(* CoDeSys 2.3.9.50 project: 152_1sha1.pro *)
(* Libraries: STANDARD.LIB 4.10.05 11:14:46, TcBase.lib 14.5.09 12:14:08, TcSystem.lib 7.6.16 11:01:22, TcUtilities.lib 16.7.20 16:08:25, SysLibVisu.lib 7.7.04 18:17:22, SysLibTargetVisu.lib 16.6.08 16:24:26, Util.lib 18.5.10 15:14:28 *)

(* Task configuration *)
TASK Standard (PRIORITY := 0, INTERVAL := T#10ms);
	MAIN
END_TASK
TASK VISU_TASK (PRIORITY := 3, INTERVAL := T#200ms);
	MAINTARGETVISU_PAINT_CODE
END_TASK
TASK VISU_INPUT_TASK (PRIORITY := 2, INTERVAL := T#50ms);
	MAINTARGETVISU_INPUT_CODE
END_TASK

(* Global variable list: Global_Variables *)
VAR_GLOBAL
(*---------------- ЛАМПЫ -------------------*)

	K152_1SHA1_HL1 					AT %Q* 	: BOOL;			(* Сеть *)
	K152_1SHA1_HL2 					AT %Q* 	: BOOL;			(* Общая авария / авария сети *)

(*----------------СОСТОЯНИЕ АВТОМАТОВ -----------------*)

	K152_1SHA1_QF1 							AT %I* 		: BOOL;		(* Положение автоматического выключателя QF1 *)
	K152_1SHA1_SF3 							AT %I* 		: BOOL;		(* Положение автоматического выключателя SF3 *)

(*----------------РАБОТА БП----------------*)

	masTABLE_POWER 							: ARRAY [1..25] OF TABLE_POWER;

	WORK_BP 									AT %I*		: BOOL;		(* Работа БП *)
	WORK_IBP 								AT %I*		: BOOL;		(* Работа ИБП *)
	WORK_OF_BATTERY 						AT %I*		: BOOL;		(* Работа от батареи *)
	REPLACE_BATTERY 						AT %I*		: BOOL;		(* Замените батарею *)

	K152_1SHA1_WORK_BP 					AT %Q*		: BOOL;		(* Работа БП *)
	K152_1SHA1_WORK_IBP 					AT %Q*		: BOOL;		(* Работа ИБП *)
	K152_1SHA1_WORK_OF_BATTERY 		AT %Q*		: BOOL;		(* Работа от батареи *)
	K152_1SHA1_REPLACE_BATTERY 			AT %Q*		: BOOL;		(* Замените батарею *)

(*---------------- ЩАО1 ----------------*)

	K152_1SHA1_SCHAO1_POWER			AT %I*		: BOOL;		(* Наличие напряжения на вводе *)
	K152_1SHA1_SCHAO1_QF1				AT %I*		: BOOL;		(* Включен автоматический выключатель QF1 *)
	K152_1SHA1_SCHAO1_QF2				AT %I*		: BOOL;		(* Включен автоматический выключатель QF2 *)
	K152_1SHA1_SCHAO1_QF3				AT %I*		: BOOL;		(* Включен автоматический выключатель QF3 *)
	K152_1SHA1_SCHAO1_QF4				AT %I*		: BOOL;		(* Включен автоматический выключатель QF4 *)
	K152_1SHA1_SCHAO1_QF5				AT %I*		: BOOL;		(* Включен автоматический выключатель QF5 *)
	K152_1SHA1_SCHAO1_QF6				AT %I*		: BOOL;		(* Включен автоматический выключатель QF6 *)
	K152_1SHA1_SCHAO1_QF7				AT %I*		: BOOL;		(* Включен автоматический выключатель QF7 *)

	K152_1SHA1_SCHAO1_KM_GR5			AT %I*		: BOOL;		(* Положение магнитного пускателя гр.5 *)

	K152_1SHA1_SCHAO1_SA_AVT_GR5		AT %I*		: BOOL;		(* Положение переключателя в режиме Авт. гр.5 *)
	K152_1SHA1_SCHAO1_SA_RUCH_GR5		AT %I*		: BOOL;		(* ?????	СМ	СХЕМУ		???????? Положение переключателя в режиме Руч. гр.5 *)

	bK152_1SHA1_SCHAO1_LIGHT_GR5_ON				: BOOL;		(* Кнопка включения группы освещения. гр.5 *)
	bK152_1SHA1_SCHAO1_LIGHT_GR5_OFF				: BOOL;		(* Кнопка выключения группы освещения. гр.5 *)
	K152_1SHA1_SCHAO1_LIGHT_GR5			AT %Q*		: BOOL;		(* Сигнал на включение группы освещения. гр.5 *)

	masTABLE_SCHAO1									: ARRAY [1..11] OF TABLE_SCHAO1;

	st_SCHAO1_POWER									: STRING;		(* Наличие напряжения на вводе *)
	st_SCHAO1_QF1										: STRING;		(* Включен автоматический выключатель QF1 *)
	st_SCHAO1_QF2										: STRING;		(* Включен автоматический выключатель QF2 *)
	st_SCHAO1_QF3										: STRING;		(* Включен автоматический выключатель QF3 *)
	st_SCHAO1_QF4										: STRING;		(* Включен автоматический выключатель QF4 *)
	st_SCHAO1_QF5										: STRING;		(* Включен автоматический выключатель QF5 *)
	st_SCHAO1_QF6										: STRING;		(* Включен автоматический выключатель QF6 *)
	st_SCHAO1_QF7										: STRING;		(* Включен автоматический выключатель QF7 *)

	st_SCHAO1_KM_GR5									: STRING;		(* Положение магнитного пускателя гр.5 *)

	st_SCHAO1_SA_AVT_GR5								: STRING;		(* Положение переключателя в режиме Авт. гр.5 *)
	st_SCHAO1_SA_RUCH_GR5							: STRING;		(* ?????	СМ	СХЕМУ		???????? Положение переключателя в режиме Руч. гр.5 *)

	st_SCHAO1_LIGHT_GR5								: STRING;		(* Сигнал на включение группы освещения. гр.5 *)

(*---------------- ЩАО2 ----------------*)

	K152_1SHA1_SCHAO2_POWER			AT %I*		: BOOL;		(* Наличие напряжения на вводе *)
	K152_1SHA1_SCHAO2_QF1				AT %I*		: BOOL;		(* Включен автоматический выключатель QF1 *)
	K152_1SHA1_SCHAO2_QF2				AT %I*		: BOOL;		(* Включен автоматический выключатель QF2 *)
	K152_1SHA1_SCHAO2_QF3				AT %I*		: BOOL;		(* Включен автоматический выключатель QF3 *)
	K152_1SHA1_SCHAO2_QF4				AT %I*		: BOOL;		(* Включен автоматический выключатель QF4 *)
	K152_1SHA1_SCHAO2_QF5				AT %I*		: BOOL;		(* Включен автоматический выключатель QF5 *)
	K152_1SHA1_SCHAO2_QF6				AT %I*		: BOOL;		(* Включен автоматический выключатель QF6 *)
	K152_1SHA1_SCHAO2_QF7				AT %I*		: BOOL;		(* Включен автоматический выключатель QF7 *)
	K152_1SHA1_SCHAO2_QF8				AT %I*		: BOOL;		(* Включен автоматический выключатель QF8 *)
	K152_1SHA1_SCHAO2_QF9				AT %I*		: BOOL;		(* Включен автоматический выключатель QF9 *)

	K152_1SHA1_SCHAO2_KM_GR5			AT %I*		: BOOL;		(* Положение магнитного пускателя гр.5 *)

	K152_1SHA1_SCHAO2_SA_AVT_GR5		AT %I*		: BOOL;		(* Положение переключателя в режиме Авт. гр.5 *)
	K152_1SHA1_SCHAO2_SA_RUCH_GR5		AT %I*		: BOOL;		(* ?????	СМ	СХЕМУ		???????? Положение переключателя в режиме Руч. гр.5 *)

	K152_1SHA1_SCHAO2_LIGHT_GR5			AT %Q*		: BOOL;		(* Сигнал на включение группы освещения. гр.5 *)

	masTABLE_SCHAO2									: ARRAY [1..13] OF TABLE_SCHAO2;

	st_SCHAO2_POWER									: STRING;		(* Наличие напряжения на вводе *)
	st_SCHAO2_QF1										: STRING;		(* Включен автоматический выключатель QF1 *)
	st_SCHAO2_QF2										: STRING;		(* Включен автоматический выключатель QF2 *)
	st_SCHAO2_QF3										: STRING;		(* Включен автоматический выключатель QF3 *)
	st_SCHAO2_QF4										: STRING;		(* Включен автоматический выключатель QF4 *)
	st_SCHAO2_QF5										: STRING;		(* Включен автоматический выключатель QF5 *)
	st_SCHAO2_QF6										: STRING;		(* Включен автоматический выключатель QF6 *)
	st_SCHAO2_QF7										: STRING;		(* Включен автоматический выключатель QF7 *)
	st_SCHAO2_QF8										: STRING;		(* Включен автоматический выключатель QF8 *)
	st_SCHAO2_QF9										: STRING;		(* Включен автоматический выключатель QF9 *)

	st_SCHAO2_KM_GR5									: STRING;		(* Положение магнитного пускателя гр.5 *)

	st_SCHAO2_SA_AVT_GR5								: STRING;		(* Положение переключателя в режиме Авт. гр.5 *)
	st_SCHAO2_SA_RUCH_GR5							: STRING;		(* ?????	СМ	СХЕМУ		???????? Положение переключателя в режиме Руч. гр.5 *)

	st_SCHAO2_LIGHT_GR5								: STRING;		(* Сигнал на включение группы освещения. гр.5 *)

	bK152_1SHA1_SCHAO2_LIGHT_GR5_ON				: BOOL;		(* Кнопка включения группы освещения. гр.5 *)
	bK152_1SHA1_SCHAO2_LIGHT_GR5_OFF				: BOOL;		(* Кнопка выключения группы освещения. гр.5 *)

(*---------------- ЩО1 ----------------*)

	K152_1SHA1_SCHO1_QF1					AT %I*		: BOOL;		(* Включен автоматический выключатель QF1 *)
	K152_1SHA1_SCHO1_QF2					AT %I*		: BOOL;		(* Включен автоматический выключатель QF2 *)

	K152_1SHA1_SCHO1_KM_GR1				AT %I*		: BOOL;		(* Положение магнитного пускателя гр.1 *)
	K152_1SHA1_SCHO1_KM_GR2				AT %I*		: BOOL;		(* Положение магнитного пускателя гр.2 *)

	K152_1SHA1_SCHO1_SA_AVT_GR1		AT %I*		: BOOL;		(* Положение переключателя в режиме Авт. гр.1 *)
	K152_1SHA1_SCHO1_SA_AVT_GR2		AT %I*		: BOOL;		(* Положение переключателя в режиме Авт. гр.2 *)

	K152_1SHA1_SCHO1_SA_RUCH_GR1		AT %I*		: BOOL;		(* Положение переключателя в режиме Руч. гр.1 *)
	K152_1SHA1_SCHO1_SA_RUCH_GR2		AT %I*		: BOOL;		(* Положение переключателя в режиме Руч. гр.2 *)

	K152_1SHA1_SCHO1_LIGHT_GR1			AT %Q*		: BOOL;		(* Сигнал на включение группы освещения. гр.1 *)
	K152_1SHA1_SCHO1_LIGHT_GR2			AT %Q*		: BOOL;		(* Сигнал на включение группы освещения. гр.2 *)

	masTABLE_SCHO1										: ARRAY [1..8] OF TABLE_SCHO1;

	st_SCHO1_QF1											: STRING;		(* Включен автоматический выключатель QF1 *)
	st_SCHO1_QF2											: STRING;		(* Включен автоматический выключатель QF2 *)

	st_SCHO1_KM_GR1									: STRING;		(* Положение магнитного пускателя гр.1 *)
	st_SCHO1_KM_GR2									: STRING;		(* Положение магнитного пускателя гр.2 *)

	st_SCHO1_SA_AVT_GR1								: STRING;		(* Положение переключателя в режиме Авт. гр.1 *)
	st_SCHO1_SA_AVT_GR2								: STRING;		(* Положение переключателя в режиме Авт. гр.2 *)

	st_SCHO1_SA_RUCH_GR1								: STRING;		(* Положение переключателя в режиме Руч. гр.1 *)
	st_SCHO1_SA_RUCH_GR2								: STRING;		(* Положение переключателя в режиме Руч. гр.2 *)

	st_SCHO1_LIGHT_GR1									: STRING;		(* Сигнал на включение группы освещения. гр.1 *)
	st_SCHO1_LIGHT_GR2									: STRING;		(* Сигнал на включение группы освещения. гр.2 *)

	bK152_1SHA1_SCHO1_LIGHT_GR1_ON					: BOOL;		(* Кнопка включения группы освещения. гр.1 *)
	bK152_1SHA1_SCHO1_LIGHT_GR2_ON					: BOOL;		(* Кнопка включения группы освещения. гр.2 *)
	bK152_1SHA1_SCHO1_LIGHT_GR1_OFF				: BOOL;		(* Кнопка выключения группы освещения. гр.1 *)
	bK152_1SHA1_SCHO1_LIGHT_GR2_OFF				: BOOL;		(* Кнопка выключения группы освещения. гр.2 *)

(*---------------- ЩО2 ----------------*)

	K152_1SHA1_SCHO2_QF1					AT %I*		: BOOL;		(* Включен автоматический выключатель QF1 *)
	K152_1SHA1_SCHO2_QF2					AT %I*		: BOOL;		(* Включен автоматический выключатель QF2 *)
	K152_1SHA1_SCHO2_QF3					AT %I*		: BOOL;		(* Включен автоматический выключатель QF3 *)
	K152_1SHA1_SCHO2_QF4					AT %I*		: BOOL;		(* Включен автоматический выключатель QF4 *)
	K152_1SHA1_SCHO2_QF5					AT %I*		: BOOL;		(* Включен автоматический выключатель QF5 *)
	K152_1SHA1_SCHO2_QF9					AT %I*		: BOOL;		(* Включен автоматический выключатель QF9 *)

	K152_1SHA1_SCHO2_KM_GR1				AT %I*		: BOOL;		(* Положение магнитного пускателя гр.1 *)
	K152_1SHA1_SCHO2_KM_GR2				AT %I*		: BOOL;		(* Положение магнитного пускателя гр.2 *)
	K152_1SHA1_SCHO2_KM_GR3				AT %I*		: BOOL;		(* Положение магнитного пускателя гр.3 *)
	K152_1SHA1_SCHO2_KM_GR4				AT %I*		: BOOL;		(* Положение магнитного пускателя гр.4 *)
	K152_1SHA1_SCHO2_KM_GR5				AT %I*		: BOOL;		(* Положение магнитного пускателя гр.5 *)
	K152_1SHA1_SCHO2_KM_GR9				AT %I*		: BOOL;		(* Положение магнитного пускателя гр.9 *)

	K152_1SHA1_SCHO2_SA_AVT_GR1		AT %I*		: BOOL;		(* Положение переключателя в режиме Авт. гр.1 *)
	K152_1SHA1_SCHO2_SA_AVT_GR2		AT %I*		: BOOL;		(* Положение переключателя в режиме Авт. гр.2 *)
	K152_1SHA1_SCHO2_SA_AVT_GR3		AT %I*		: BOOL;		(* Положение переключателя в режиме Авт. гр.3 *)
	K152_1SHA1_SCHO2_SA_AVT_GR4		AT %I*		: BOOL;		(* Положение переключателя в режиме Авт. гр.4 *)
	K152_1SHA1_SCHO2_SA_AVT_GR5		AT %I*		: BOOL;		(* Положение переключателя в режиме Авт. гр.5 *)
	K152_1SHA1_SCHO2_SA_AVT_GR9		AT %I*		: BOOL;		(* Положение переключателя в режиме Авт. гр.9 *)

	K152_1SHA1_SCHO2_SA_RUCH_GR1		AT %I*		: BOOL;		(* Положение переключателя в режиме Руч. гр.1 *)
	K152_1SHA1_SCHO2_SA_RUCH_GR2		AT %I*		: BOOL;		(* Положение переключателя в режиме Руч. гр.2 *)
	K152_1SHA1_SCHO2_SA_RUCH_GR3		AT %I*		: BOOL;		(* Положение переключателя в режиме Руч. гр.3 *)
	K152_1SHA1_SCHO2_SA_RUCH_GR4		AT %I*		: BOOL;		(* Положение переключателя в режиме Руч. гр.4 *)
	K152_1SHA1_SCHO2_SA_RUCH_GR5		AT %I*		: BOOL;		(* Положение переключателя в режиме Руч. гр.5 *)
	K152_1SHA1_SCHO2_SA_RUCH_GR9		AT %I*		: BOOL;		(* Положение переключателя в режиме Руч. гр.9 *)

	K152_1SHA1_SCHO2_LIGHT_GR1			AT %Q*		: BOOL;		(* Сигнал на включение группы освещения. гр.1 *)
	K152_1SHA1_SCHO2_LIGHT_GR2			AT %Q*		: BOOL;		(* Сигнал на включение группы освещения. гр.2 *)
	K152_1SHA1_SCHO2_LIGHT_GR3			AT %Q*		: BOOL;		(* Сигнал на включение группы освещения. гр.3 *)
	K152_1SHA1_SCHO2_LIGHT_GR4			AT %Q*		: BOOL;		(* Сигнал на включение группы освещения. гр.4 *)
	K152_1SHA1_SCHO2_LIGHT_GR5			AT %Q*		: BOOL;		(* Сигнал на включение группы освещения. гр.5 *)
	K152_1SHA1_SCHO2_LIGHT_GR9			AT %Q*		: BOOL;		(* Сигнал на включение группы освещения. гр.9 *)

	masTABLE_SCHO2_1									: ARRAY [1..4] OF TABLE;
	masTABLE_SCHO2_2									: ARRAY [1..4] OF TABLE_SCHO2;
	masTABLE_SCHO2_3									: ARRAY [1..4] OF TABLE_SCHO2;
	masTABLE_SCHO2_4									: ARRAY [1..4] OF TABLE_SCHO2;
	masTABLE_SCHO2_5									: ARRAY [1..4] OF TABLE_SCHO2;
	masTABLE_SCHO2_9									: ARRAY [1..4] OF TABLE_SCHO2;

	st_SCHO2_QF1											: STRING;		(* Включен автоматический выключатель QF1 *)
	st_SCHO2_QF2											: STRING;		(* Включен автоматический выключатель QF2 *)
	st_SCHO2_QF3											: STRING;		(* Включен автоматический выключатель QF3 *)
	st_SCHO2_QF4											: STRING;		(* Включен автоматический выключатель QF4 *)
	st_SCHO2_QF5											: STRING;		(* Включен автоматический выключатель QF5 *)
	st_SCHO2_QF9											: STRING;		(* Включен автоматический выключатель QF9 *)

	st_SCHO2_KM_GR1									: STRING;		(* Положение магнитного пускателя гр.1 *)
	st_SCHO2_KM_GR2									: STRING;		(* Положение магнитного пускателя гр.2 *)
	st_SCHO2_KM_GR3									: STRING;		(* Положение магнитного пускателя гр.3 *)
	st_SCHO2_KM_GR4									: STRING;		(* Положение магнитного пускателя гр.4 *)
	st_SCHO2_KM_GR5									: STRING;		(* Положение магнитного пускателя гр.5 *)
	st_SCHO2_KM_GR9									: STRING;		(* Положение магнитного пускателя гр.9 *)

	st_SCHO2_SA_AVT_GR1								: STRING;		(* Положение переключателя в режиме Авт. гр.1 *)
	st_SCHO2_SA_AVT_GR2								: STRING;		(* Положение переключателя в режиме Авт. гр.2 *)
	st_SCHO2_SA_AVT_GR3								: STRING;		(* Положение переключателя в режиме Авт. гр.3 *)
	st_SCHO2_SA_AVT_GR4								: STRING;		(* Положение переключателя в режиме Авт. гр.4 *)
	st_SCHO2_SA_AVT_GR5								: STRING;		(* Положение переключателя в режиме Авт. гр.5 *)
	st_SCHO2_SA_AVT_GR9								: STRING;		(* Положение переключателя в режиме Авт. гр.9 *)

	st_SCHO2_SA_RUCH_GR1								: STRING;		(* Положение переключателя в режиме Руч. гр.1 *)
	st_SCHO2_SA_RUCH_GR2								: STRING;		(* Положение переключателя в режиме Руч. гр.2 *)
	st_SCHO2_SA_RUCH_GR3								: STRING;		(* Положение переключателя в режиме Руч. гр.3 *)
	st_SCHO2_SA_RUCH_GR4								: STRING;		(* Положение переключателя в режиме Руч. гр.4 *)
	st_SCHO2_SA_RUCH_GR5								: STRING;		(* Положение переключателя в режиме Руч. гр.5 *)
	st_SCHO2_SA_RUCH_GR9								: STRING;		(* Положение переключателя в режиме Руч. гр.9 *)

	st_SCHO2_LIGHT_GR1									: STRING;		(* Сигнал на включение группы освещения. гр.1 *)
	st_SCHO2_LIGHT_GR2									: STRING;		(* Сигнал на включение группы освещения. гр.2 *)
	st_SCHO2_LIGHT_GR3									: STRING;		(* Сигнал на включение группы освещения. гр.3 *)
	st_SCHO2_LIGHT_GR4									: STRING;		(* Сигнал на включение группы освещения. гр.4 *)
	st_SCHO2_LIGHT_GR5									: STRING;		(* Сигнал на включение группы освещения. гр.5 *)
	st_SCHO2_LIGHT_GR9									: STRING;		(* Сигнал на включение группы освещения. гр.9 *)

	bK152_1SHA1_SCHO2_LIGHT_GR1_ON					: BOOL;		(* Кнопка включения группы освещения. гр.1 *)
	bK152_1SHA1_SCHO2_LIGHT_GR2_ON					: BOOL;		(* Кнопка включения группы освещения. гр.2 *)
	bK152_1SHA1_SCHO2_LIGHT_GR3_ON					: BOOL;		(* Кнопка включения группы освещения. гр.3 *)
	bK152_1SHA1_SCHO2_LIGHT_GR4_ON					: BOOL;		(* Кнопка включения группы освещения. гр.4 *)
	bK152_1SHA1_SCHO2_LIGHT_GR5_ON					: BOOL;		(* Кнопка включения группы освещения. гр.5 *)
	bK152_1SHA1_SCHO2_LIGHT_GR9_ON					: BOOL;		(* Кнопка включения группы освещения. гр.9 *)

	bK152_1SHA1_SCHO2_LIGHT_GR1_OFF				: BOOL;		(* Кнопка выключения группы освещения. гр.1 *)
	bK152_1SHA1_SCHO2_LIGHT_GR2_OFF				: BOOL;		(* Кнопка выключения группы освещения. гр.2 *)
	bK152_1SHA1_SCHO2_LIGHT_GR3_OFF				: BOOL;		(* Кнопка выключения группы освещения. гр.3 *)
	bK152_1SHA1_SCHO2_LIGHT_GR4_OFF				: BOOL;		(* Кнопка выключения группы освещения. гр.4 *)
	bK152_1SHA1_SCHO2_LIGHT_GR5_OFF				: BOOL;		(* Кнопка выключения группы освещения. гр.5 *)
	bK152_1SHA1_SCHO2_LIGHT_GR9_OFF				: BOOL;		(* Кнопка выключения группы освещения. гр.9 *)

(* 	Режимы работы *)
	K152_1SHA1_SCHO2_GR1_bMode		 				: BOOL;		(* Выбор режима управления Группой 1 *)
	K152_1SHA1_SCHO2_GR1_Mode		 				: STRING;		(* Режим управления Группой 1 *)

	Invisible_GR1_bMode									: BOOL;		(* Невидимость кнопок выбора режима Гр.1 *)
	Invisible_GR1_bMode_MU								: BOOL;		(* Невидимость кнопок управления руч. режима Гр.1 *)


	K152_1SHA1_SCHO2_GR1_bMode_AVT 				: BOOL;		(* Режим автоматического управления Группой 1 *)
	K152_1SHA1_SCHO2_GR2_bMode_AVT 				: BOOL;		(* Режим автоматического управления Группой 2 *)
	K152_1SHA1_SCHO2_GR3_bMode_AVT 				: BOOL;		(* Режим автоматического управления Группой 3 *)
	K152_1SHA1_SCHO2_GR4_bMode_AVT 				: BOOL;		(* Режим автоматического управления Группой 4 *)
	K152_1SHA1_SCHO2_GR5_bMode_AVT 				: BOOL;		(* Режим автоматического управления Группой 5 *)
	K152_1SHA1_SCHO2_GR9_bMode_AVT 				: BOOL;		(* Режим автоматического управления Группой 9 *)

	K152_1SHA1_SCHO2_GR1_bMode_MU	 				: BOOL;		(* Режим ручного управления Группой 1 *)
	K152_1SHA1_SCHO2_GR2_bMode_MU	 				: BOOL;		(* Режим ручного управления Группой 2 *)
	K152_1SHA1_SCHO2_GR3_bMode_MU	 				: BOOL;		(* Режим ручного управления Группой 3 *)
	K152_1SHA1_SCHO2_GR4_bMode_MU	 				: BOOL;		(* Режим ручного управления Группой 4 *)
	K152_1SHA1_SCHO2_GR5_bMode_MU	 				: BOOL;		(* Режим ручного управления Группой 5 *)
	K152_1SHA1_SCHO2_GR9_bMode_MU	 				: BOOL;		(* Режим ручного управления Группой 9 *)

(* 	Недельный график *)
	masTABLE_WEEKLY_SCHO2_GR1						: ARRAY [1..2] OF TABLE_WEEKLY_SCHEDULE;

(*---------------- Датчики протечки ----------------*)

	K152_1SHA1_LS_ITP_1						AT %I*		: BOOL;		(* Датчик протечки LS-ИТП-1 *)
	K152_1SHA1_LS_ITP_2						AT %I*		: BOOL;		(* Датчик протечки LS-ИТП-2 *)
	K152_1SHA1_LS_NS_1						AT %I*		: BOOL;		(* Датчик протечки LS-НС-1 *)
	K152_1SHA1_LS_NS_2						AT %I*		: BOOL;		(* Датчик протечки LS-НС-2 *)

(*---------------- Коробка соединительная КС1 ----------------*)

	K152_1SHA1_KC1_BK1_TRESH1			AT %I*		: BOOL;		(* Блок контроля 1, Срабатывание порога 1 *)
	K152_1SHA1_KC1_BK2_TRESH1			AT %I*		: BOOL;		(* Блок контроля 2, Срабатывание порога 1 *)
	K152_1SHA1_KC1_BK3_TRESH1			AT %I*		: BOOL;		(* Блок контроля 3, Срабатывание порога 1 *)
	K152_1SHA1_KC1_BK4_TRESH1			AT %I*		: BOOL;		(* Блок контроля 4, Срабатывание порога 1 *)

	K152_1SHA1_KC1_BK1_TRESH2			AT %I*		: BOOL;		(* Блок контроля 1, Срабатывание порога 2 *)
	K152_1SHA1_KC1_BK2_TRESH2			AT %I*		: BOOL;		(* Блок контроля 2, Срабатывание порога 2 *)
	K152_1SHA1_KC1_BK3_TRESH2			AT %I*		: BOOL;		(* Блок контроля 3, Срабатывание порога 2 *)
	K152_1SHA1_KC1_BK4_TRESH2			AT %I*		: BOOL;		(* Блок контроля 4, Срабатывание порога 2 *)

	K152_1SHA1_KC1_BLIND_CLOSE			AT %Q*		: BOOL;		(* Сигнал на закрытие жалюзи помещение 1.4.2 *)
	K152_1SHA1_KC1_BLIND_OPEN			AT %Q*		: BOOL;		(* Сигнал на открытие жалюзи помещение 1.4.2 *)

(*---------------- Коробка соединительная КС2 ----------------*)

	K152_1SHA1_KC2_BLIND_CLOSE			AT %Q*		: BOOL;		(* Сигнал на закрытие жалюзи помещение 1.4.1 *)
	K152_1SHA1_KC2_BLIND_OPEN			AT %Q*		: BOOL;		(* Сигнал на открытие жалюзи помещение 1.4.1 *)

(*---------------- Коробка соединительная КС3 ----------------*)

	K152_1SHA1_KC3_BLIND_CLOSE			AT %Q*		: BOOL;		(* Сигнал на закрытие жалюзи помещение 1.4.0 *)
	K152_1SHA1_KC3_BLIND_OPEN			AT %Q*		: BOOL;		(* Сигнал на открытие жалюзи помещение 1.4.0 *)

(*---------------- ШРС ----------------*)

	K152_1SHA1_WORK_ALARM_MEDOMAT	AT %I*		: BOOL;		(* Контроль работы / аварии установки Medomat *)
	K152_1SHA1_WORK_ALARM_FILTER1		AT %I*		: BOOL;		(* Контроль работы / аварии фильтра обезжелезивания 1 *)
	K152_1SHA1_WORK_ALARM_FILTER2		AT %I*		: BOOL;		(* Контроль работы / аварии фильтра обезжелезивания 2 *)
	K152_1SHA1_WORK_ALARM_RONDOMAT	AT %I*		: BOOL;		(* Контроль работы / аварии установки Rondomat *)

 	K152_1SHA1_LEVEL_TANK1				AT %I*		: BOOL;		(* Контроль уровня жидкости в резервуре 1 *)
 	K152_1SHA1_LEVEL_TANK2				AT %I*		: BOOL;		(* Контроль уровня жидкости в резервуре 2 *)
 	K152_1SHA1_LEVEL_TANK3				AT %I*		: BOOL;		(* Контроль уровня жидкости в резервуре 3 *)
 	K152_1SHA1_LEVEL_TANK4				AT %I*		: BOOL;		(* Контроль уровня жидкости в резервуре 4 *)
 	K152_1SHA1_LEVEL_TANK5				AT %I*		: BOOL;		(* Контроль уровня жидкости в резервуре 5 *)

 	K152_1SHA1_WORK_ALARM_OSMOSIS	AT %I*		: BOOL;		(* Контроль работы / аварии установки обратного осмоса *)

(*---------------- ПКУ1 ----------------*)

	K152_1SHA1_PKU1_SA					AT %I*		: BOOL;		(* Переключатель руч. / авт. помещение 1.4.2 *)
	K152_1SHA1_PKU1_SB_CLOSE			AT %I*		: BOOL;		(* Кнопка закрыть жалюзи помещение 1.4.2 *)
	K152_1SHA1_PKU1_SB_OPEN				AT %I*		: BOOL;		(* Кнопка открыть жалюзи помещение 1.4.2 *)

(*---------------- ПКУ2 ----------------*)

	K152_1SHA1_PKU2_SA					AT %I*		: BOOL;		(* Переключатель руч. / авт. помещение 1.4.1 *)
	K152_1SHA1_PKU2_SB_CLOSE			AT %I*		: BOOL;		(* Кнопка закрыть жалюзи помещение 1.4.1 *)
	K152_1SHA1_PKU2_SB_OPEN				AT %I*		: BOOL;		(* Кнопка открыть жалюзи помещение 1.4.1 *)

(*---------------- ПКУ3 ----------------*)

	K152_1SHA1_PKU3_SA					AT %I*		: BOOL;		(* Переключатель руч. / авт. помещение 1.4.0 *)
	K152_1SHA1_PKU3_SB_CLOSE			AT %I*		: BOOL;		(* Кнопка закрыть жалюзи помещение 1.4.0 *)
	K152_1SHA1_PKU3_SB_OPEN				AT %I*		: BOOL;		(* Кнопка открыть жалюзи помещение 1.4.0 *)

(*----------------ТЕМПЕРАТУРА----------------*)

	masTABLE_TEMPERATURE					: ARRAY [1..10] OF TABLE_TEMPERATURE;

	TE_TK 										AT %I*		: INT;			(* Температура воздуха в ТК, TE-TK *)
	TE_GRSCHA 								AT %I*		: INT;			(* Температура воздуха в ГРЩ TE-ГРЩ *)

	K152_1SHA1_TE_TK 						AT %Q*		: REAL;			(* Температура воздуха в ТК, TE-TK *)
	K152_1SHA1_TE_GRSCHA					AT %Q*		: REAL;			(* Температура воздуха в ГРЩ, TE-ГРЩ *)


(* --------------------- СИСТЕМНОЕ ДАТА И ВРЕМЯ -------------------------- *)
	stDate 													: STRING;		(* Текущая дата *)
	stTime 													: STRING;		(* Текущее время *)
	stTime_graphic											: STRING;		(* Часы и минуты для недельного графика *)

	Day_of_Today											: STRING;		(* Текущий день недели *)
(* --------------------- ТАБЛИЦА АВАРИЙ -------------------------- *)

	(* Дата и время *)
	stTime_Alarm											: STRING;
	stDate_Alarm											: STRING;

	(* --------------------- *)
(*
	rt_K152_1ITP_K1 								: R_TRIG ;			(* Авария входного напряжения *)
	ft_K152_1ITP_1PDS1 							: F_TRIG;			(* Перепад давления в системе отопления *)
	ft_K152_1ITP_2PDS1 							: F_TRIG;			(* Перепад давления в системе ГВС *)
	ft_K152_1ITP_2PDS2 							: F_TRIG;			(* Перепад давления в системе вентиляции *)
	ft_K152_1ITP_2PDS3 							: F_TRIG;			(* Перепад давления в системе подпитки вентиляции *)
	rt_K152_1ITP_QF1_ALARM 						: R_TRIG;
	rt_K152_1ITP_QF2_ALARM 						: R_TRIG;
	rt_K152_1ITP_QF3_ALARM	 					: R_TRIG;
	rt_K152_1ITP_QF4_ALARM 						: R_TRIG;
	rt_K152_1ITP_QF5_ALARM 						: R_TRIG;
	rt_K152_1ITP_QF6_ALARM 						: R_TRIG;
	rt_K152_1ITP_QF7_ALARM 						: R_TRIG;
	rt_K152_1ITP_QF8_ALARM 						: R_TRIG;

	rt_K152_1ITP_REPLACE_BATTERY				: R_TRIG;

	rt_K152_1ITP_UPK_ALARM 					: R_TRIG;			(* Авария установки перекачки конденсата *)
	rt_K152_1ITP_LS 								: R_TRIG;			(* Низкий уровень воды в баке ресивере *)

	rt_K152_1ITP_HL4 								: R_TRIG;			(* Авария основного насоса 2.1 *)
	rt_K152_1ITP_HL6 								: R_TRIG;			(* Авария резервного насоса 2.2 *)
	rt_K152_1ITP_HL8 								: R_TRIG;			(* Авария основного насоса 6.1 *)
	rt_K152_1ITP_HL10 								: R_TRIG;			(* Авария резервного насоса 6.2 *)
	rt_K152_1ITP_HL12 								: R_TRIG;			(* Авария основного насоса 7.1 *)
	rt_K152_1ITP_HL14 								: R_TRIG;			(* Авария резервного насоса 7.2 *)
	rt_K152_1ITP_HL16 								: R_TRIG;			(* Авария основного насоса 12.1 *)
	rt_K152_1ITP_HL18 								: R_TRIG;			(* Авария резервного насоса 12.2 *)
*)
	i 												: INT 	:= 	0;		(* Счетчик строк в таблице аварий *)
	d 												: INT 	:= 	0;		(* Счетчик записей в массив данных об авариях *)

	ALARM_TABLE 								: ARRAY [1..23] OF TABLE_ALARM;
	ALARM_DATA 									: ARRAY [1..100] OF STRING;					(* Запись инфо об аварии в одну переменную *)

	bClearAlarmData 								: BOOL;
	rt_bClearAlarmData								: R_TRIG;

END_VAR

(* Global variable list: TwinCAT_Configuration *)
(* Generated automatically by TwinCAT - (read only) *)
VAR_CONFIG
	.K152_1SHA1_HL1 AT %QX12.0 : BOOL;
	.K152_1SHA1_HL2 AT %QX12.1 : BOOL;
	.K152_1SHA1_QF1 AT %IX4.0 : BOOL;
	.K152_1SHA1_SF3 AT %IX4.1 : BOOL;
	.WORK_BP AT %IX4.2 : BOOL;
	.WORK_IBP AT %IX4.3 : BOOL;
	.WORK_OF_BATTERY AT %IX4.4 : BOOL;
	.REPLACE_BATTERY AT %IX4.5 : BOOL;
	.K152_1SHA1_WORK_BP AT %QX8.0 : BOOL;
	.K152_1SHA1_WORK_IBP AT %QX8.1 : BOOL;
	.K152_1SHA1_WORK_OF_BATTERY AT %QX8.2 : BOOL;
	.K152_1SHA1_REPLACE_BATTERY AT %QX8.3 : BOOL;
	.K152_1SHA1_SCHAO1_POWER AT %IX4.6 : BOOL;
	.K152_1SHA1_SCHAO1_QF1 AT %IX4.7 : BOOL;
	.K152_1SHA1_SCHAO1_QF2 AT %IX5.0 : BOOL;
	.K152_1SHA1_SCHAO1_QF3 AT %IX5.1 : BOOL;
	.K152_1SHA1_SCHAO1_QF4 AT %IX5.2 : BOOL;
	.K152_1SHA1_SCHAO1_QF5 AT %IX5.3 : BOOL;
	.K152_1SHA1_SCHAO1_QF6 AT %IX5.4 : BOOL;
	.K152_1SHA1_SCHAO1_QF7 AT %IX5.5 : BOOL;
	.K152_1SHA1_SCHAO1_KM_GR5 AT %IX5.6 : BOOL;
	.K152_1SHA1_SCHAO1_SA_AVT_GR5 AT %IX5.7 : BOOL;
	.K152_1SHA1_SCHAO1_SA_RUCH_GR5 AT %IX6.0 : BOOL;
	.K152_1SHA1_SCHAO1_LIGHT_GR5 AT %QX8.4 : BOOL;
	.K152_1SHA1_SCHAO2_POWER AT %IX6.1 : BOOL;
	.K152_1SHA1_SCHAO2_QF1 AT %IX6.2 : BOOL;
	.K152_1SHA1_SCHAO2_QF2 AT %IX6.3 : BOOL;
	.K152_1SHA1_SCHAO2_QF3 AT %IX6.4 : BOOL;
	.K152_1SHA1_SCHAO2_QF4 AT %IX6.5 : BOOL;
	.K152_1SHA1_SCHAO2_QF5 AT %IX6.6 : BOOL;
	.K152_1SHA1_SCHAO2_QF6 AT %IX6.7 : BOOL;
	.K152_1SHA1_SCHAO2_QF7 AT %IX7.0 : BOOL;
	.K152_1SHA1_SCHAO2_QF8 AT %IX7.1 : BOOL;
	.K152_1SHA1_SCHAO2_QF9 AT %IX7.2 : BOOL;
	.K152_1SHA1_SCHAO2_KM_GR5 AT %IX7.3 : BOOL;
	.K152_1SHA1_SCHAO2_SA_AVT_GR5 AT %IX7.4 : BOOL;
	.K152_1SHA1_SCHAO2_SA_RUCH_GR5 AT %IX7.5 : BOOL;
	.K152_1SHA1_SCHAO2_LIGHT_GR5 AT %QX8.5 : BOOL;
	.K152_1SHA1_SCHO1_QF1 AT %IX7.6 : BOOL;
	.K152_1SHA1_SCHO1_QF2 AT %IX7.7 : BOOL;
	.K152_1SHA1_SCHO1_KM_GR1 AT %IX8.0 : BOOL;
	.K152_1SHA1_SCHO1_KM_GR2 AT %IX8.1 : BOOL;
	.K152_1SHA1_SCHO1_SA_AVT_GR1 AT %IX8.2 : BOOL;
	.K152_1SHA1_SCHO1_SA_AVT_GR2 AT %IX8.3 : BOOL;
	.K152_1SHA1_SCHO1_SA_RUCH_GR1 AT %IX8.4 : BOOL;
	.K152_1SHA1_SCHO1_SA_RUCH_GR2 AT %IX8.5 : BOOL;
	.K152_1SHA1_SCHO1_LIGHT_GR1 AT %QX8.6 : BOOL;
	.K152_1SHA1_SCHO1_LIGHT_GR2 AT %QX8.7 : BOOL;
	.K152_1SHA1_SCHO2_QF1 AT %IX8.6 : BOOL;
	.K152_1SHA1_SCHO2_QF2 AT %IX8.7 : BOOL;
	.K152_1SHA1_SCHO2_QF3 AT %IX9.0 : BOOL;
	.K152_1SHA1_SCHO2_QF4 AT %IX9.1 : BOOL;
	.K152_1SHA1_SCHO2_QF5 AT %IX9.2 : BOOL;
	.K152_1SHA1_SCHO2_QF9 AT %IX9.3 : BOOL;
	.K152_1SHA1_SCHO2_KM_GR1 AT %IX9.4 : BOOL;
	.K152_1SHA1_SCHO2_KM_GR2 AT %IX9.5 : BOOL;
	.K152_1SHA1_SCHO2_KM_GR3 AT %IX9.6 : BOOL;
	.K152_1SHA1_SCHO2_KM_GR4 AT %IX9.7 : BOOL;
	.K152_1SHA1_SCHO2_KM_GR5 AT %IX10.0 : BOOL;
	.K152_1SHA1_SCHO2_KM_GR9 AT %IX10.1 : BOOL;
	.K152_1SHA1_SCHO2_SA_AVT_GR1 AT %IX10.2 : BOOL;
	.K152_1SHA1_SCHO2_SA_AVT_GR2 AT %IX10.3 : BOOL;
	.K152_1SHA1_SCHO2_SA_AVT_GR3 AT %IX10.4 : BOOL;
	.K152_1SHA1_SCHO2_SA_AVT_GR4 AT %IX10.5 : BOOL;
	.K152_1SHA1_SCHO2_SA_AVT_GR5 AT %IX10.6 : BOOL;
	.K152_1SHA1_SCHO2_SA_AVT_GR9 AT %IX10.7 : BOOL;
	.K152_1SHA1_SCHO2_SA_RUCH_GR1 AT %IX11.0 : BOOL;
	.K152_1SHA1_SCHO2_SA_RUCH_GR2 AT %IX11.1 : BOOL;
	.K152_1SHA1_SCHO2_SA_RUCH_GR3 AT %IX11.2 : BOOL;
	.K152_1SHA1_SCHO2_SA_RUCH_GR4 AT %IX11.3 : BOOL;
	.K152_1SHA1_SCHO2_SA_RUCH_GR5 AT %IX11.4 : BOOL;
	.K152_1SHA1_SCHO2_SA_RUCH_GR9 AT %IX11.5 : BOOL;
	.K152_1SHA1_SCHO2_LIGHT_GR1 AT %QX9.0 : BOOL;
	.K152_1SHA1_SCHO2_LIGHT_GR2 AT %QX9.1 : BOOL;
	.K152_1SHA1_SCHO2_LIGHT_GR3 AT %QX9.2 : BOOL;
	.K152_1SHA1_SCHO2_LIGHT_GR4 AT %QX9.3 : BOOL;
	.K152_1SHA1_SCHO2_LIGHT_GR5 AT %QX9.4 : BOOL;
	.K152_1SHA1_SCHO2_LIGHT_GR9 AT %QX9.5 : BOOL;
	.K152_1SHA1_LS_ITP_1 AT %IX11.6 : BOOL;
	.K152_1SHA1_LS_ITP_2 AT %IX11.7 : BOOL;
	.K152_1SHA1_LS_NS_1 AT %IX12.0 : BOOL;
	.K152_1SHA1_LS_NS_2 AT %IX12.1 : BOOL;
	.K152_1SHA1_KC1_BK1_TRESH1 AT %IX12.2 : BOOL;
	.K152_1SHA1_KC1_BK2_TRESH1 AT %IX12.3 : BOOL;
	.K152_1SHA1_KC1_BK3_TRESH1 AT %IX12.4 : BOOL;
	.K152_1SHA1_KC1_BK4_TRESH1 AT %IX12.5 : BOOL;
	.K152_1SHA1_KC1_BK1_TRESH2 AT %IX12.6 : BOOL;
	.K152_1SHA1_KC1_BK2_TRESH2 AT %IX12.7 : BOOL;
	.K152_1SHA1_KC1_BK3_TRESH2 AT %IX13.0 : BOOL;
	.K152_1SHA1_KC1_BK4_TRESH2 AT %IX13.1 : BOOL;
	.K152_1SHA1_KC1_BLIND_CLOSE AT %QX9.6 : BOOL;
	.K152_1SHA1_KC1_BLIND_OPEN AT %QX9.7 : BOOL;
	.K152_1SHA1_KC2_BLIND_CLOSE AT %QX10.0 : BOOL;
	.K152_1SHA1_KC2_BLIND_OPEN AT %QX10.1 : BOOL;
	.K152_1SHA1_KC3_BLIND_CLOSE AT %QX10.2 : BOOL;
	.K152_1SHA1_KC3_BLIND_OPEN AT %QX10.3 : BOOL;
	.K152_1SHA1_WORK_ALARM_MEDOMAT AT %IX13.2 : BOOL;
	.K152_1SHA1_WORK_ALARM_FILTER1 AT %IX13.3 : BOOL;
	.K152_1SHA1_WORK_ALARM_FILTER2 AT %IX13.4 : BOOL;
	.K152_1SHA1_WORK_ALARM_RONDOMAT AT %IX13.5 : BOOL;
	.K152_1SHA1_LEVEL_TANK1 AT %IX13.6 : BOOL;
	.K152_1SHA1_LEVEL_TANK2 AT %IX13.7 : BOOL;
	.K152_1SHA1_LEVEL_TANK3 AT %IX14.0 : BOOL;
	.K152_1SHA1_LEVEL_TANK4 AT %IX14.1 : BOOL;
	.K152_1SHA1_LEVEL_TANK5 AT %IX14.2 : BOOL;
	.K152_1SHA1_WORK_ALARM_OSMOSIS AT %IX14.3 : BOOL;
	.K152_1SHA1_PKU1_SA AT %IX14.4 : BOOL;
	.K152_1SHA1_PKU1_SB_CLOSE AT %IX14.5 : BOOL;
	.K152_1SHA1_PKU1_SB_OPEN AT %IX14.6 : BOOL;
	.K152_1SHA1_PKU2_SA AT %IX14.7 : BOOL;
	.K152_1SHA1_PKU2_SB_CLOSE AT %IX15.0 : BOOL;
	.K152_1SHA1_PKU2_SB_OPEN AT %IX15.1 : BOOL;
	.K152_1SHA1_PKU3_SA AT %IX15.2 : BOOL;
	.K152_1SHA1_PKU3_SB_CLOSE AT %IX15.3 : BOOL;
	.K152_1SHA1_PKU3_SB_OPEN AT %IX15.4 : BOOL;
	.TE_TK AT %IB0 : INT;
	.TE_GRSCHA AT %IB2 : INT;
	.K152_1SHA1_TE_TK AT %QB0 : REAL;
	.K152_1SHA1_TE_GRSCHA AT %QB4 : REAL;
END_VAR

(* Data type *)
TYPE TABLE :
STRUCT
	Position 			: STRING;		(* Узел *)
	On_Off				: STRING;		(* Текущее положение *)
	ON					: BOOL;		(* Изменение цвета в столбце *)
END_STRUCT
END_TYPE

(* Data type *)
TYPE TABLE_ALARM :
STRUCT
	s1Date : STRING;			(* Дата аварии *)
	s2Time : STRING;			(* Время аварии *)
	s3Text : STRING;			(* Текст сообщения *)
END_STRUCT
END_TYPE

(* Data type *)
TYPE TABLE_CIRCUITS :
STRUCT
	s1Text : STRING;
	s2Text : STRING;
	dwFillColorAlarm : DWORD;
END_STRUCT
END_TYPE

(* Data type *)
TYPE TABLE_POWER :
STRUCT
	s1Text : STRING;
	s2Text : STRING;
	dwFillColorAlarm : DWORD;
END_STRUCT
END_TYPE

(* Data type *)
TYPE TABLE_SCHAO1 :
STRUCT
	s1Positioin 			: STRING;		(* Узел *)
	s2Value_X			: STRING;		(* Текущее положение *)
	s3Value_SET		: REAL;			(* Управление *)
	dwFillColorAlarm 	: DWORD;
END_STRUCT
END_TYPE

(* Data type *)
TYPE TABLE_SCHAO2 :
STRUCT
	s1Positioin 			: STRING;		(* Узел *)
	s2Value_X			: STRING;		(* Текущее положение *)
	s3Value_SET		: REAL;			(* Управление *)
	dwFillColorAlarm 	: DWORD;
END_STRUCT
END_TYPE

(* Data type *)
TYPE TABLE_SCHO1 :
STRUCT
	s1Positioin 			: STRING;		(* Узел *)
	s2Value_X			: STRING;		(* Текущее положение *)
	s3Value_SET		: REAL;			(* Управление *)
	dwFillColorAlarm 	: DWORD;
END_STRUCT
END_TYPE

(* Data type *)
TYPE TABLE_SCHO2 :
STRUCT
	s1Positioin 			: STRING;		(* Узел *)
	s2Value_X			: STRING;		(* Текущее положение *)
	s3Value_SET		: REAL;			(* Управление *)
	dwFillColorAlarm 	: DWORD;
END_STRUCT
END_TYPE

(* Data type *)
TYPE TABLE_TEMPERATURE :
STRUCT
	s1Positioin 		: STRING;			(* Позиция датчика *)
	s2Value			: REAL;				(* Текущее значение *)
END_STRUCT
END_TYPE

(* Data type *)
TYPE TABLE_WEEKLY_SCHEDULE :
STRUCT
	Parameters		: STRING;			(* Столбец дня недели и времени включения / выключения *)
	s1Mon 			: STRING;			(* Столбец Понедельника *)
	s2Tues 			: STRING;			(* Столбец Вторника *)
	s3Wed	 		: STRING;			(* Столбец Среды *)
	s4Thrus 		: STRING;			(* Столбец Четверга *)
	s5Fri 			: STRING;			(* Столбец Пятницы *)
	s6Sat 			: STRING;			(* Столбец Субботы *)
	s7Sun 			: STRING;			(* Столбец Воскресенья *)
END_STRUCT
END_TYPE

(* POU MAIN, ST *)
PROGRAM MAIN
VAR
END_VAR
DATE_AND_TIME_SYSTEM();
LAMPS();
VHOD();
SCHAO1();
SCHAO2();
SCHO1();
SCHO2();
SCHO2_TABLE_OF_WEEKLY_SCHEDULE();
END_PROGRAM

(* POU DATE_AND_TIME_SYSTEM, ST *)
PROGRAM DATE_AND_TIME_SYSTEM
VAR
  	fbSystemTime    	: GETSYSTEMTIME;
    	timeAsFileTime  	: T_FILETIME;
    	timeAsDT       		: DT;
	input_date			: DATE;
	input_time			: TOD;
	real_time			: TIME;
	summa				: TIME;
	time_time			: TIME;
	now_time			: TOD;

	output_time			: STRING;
	output_date			: STRING;
	day					: STRING;
	tire					: STRING;
	month				: STRING;
	year				: STRING;
	year_not_tire		: STRING;

	conc1				: STRING;
	conc2				: STRING;

	stSumma_dt 		: ARRAY [1..100] OF STRING;				(* Записывает дату и время в одну переменную *)
	razdelitel			: STRING;
	stDate_r			: STRING;
	stTime_r			: STRING;
	stDate_and_Time	: STRING;
	stAlarm_Data		: STRING;

(*	Определние дня недели *)
	NumOfDay 			: DWORD;
	dDate 				: DATE;
	DAY_OF_WEEK 	: UINT;
END_VAR
fbSystemTime(
    timeLoDW =>timeAsFileTime.dwLowDateTime,
    timeHiDW =>timeAsFileTime.dwHighDateTime 
);
timeAsDT := FILETIME_TO_DT( timeAsFileTime );

input_time :=DT_TO_TOD(timeAsDT);		(* отделяем время от даты_и_времени *)
input_date :=DT_TO_DATE(timeAsDT);		(* отделяем дату от даты_и_времени *)

time_time :=TOD_TO_TIME(input_time);		(* преобразуем время в время *)
summa := t#03h00m00s;					(* задаем разницу в часах - 3 часа от реального времени *)
real_time := time_time + summa;			(* суммируем разницу и входное время *)

now_time := TIME_TO_TOD(real_time);			(* представляем сумму в виде дата_и_время *)

output_time := TOD_TO_STRING(now_time);			(* записываем время как тип стринг для таблицы аварий*)
output_date := DATE_TO_STRING(input_date);		(* записываем дату как тип стринг для таблицы аварий *)

day := MID(output_date, 13, 11);					(* Отделяем день *)
month := MID(output_date, 3, 7);					(* Отделяем месяц *)
year_not_tire := MID(output_date, 4, 3);			(* Отделяем год *)
tire := '-';										(* Задаем символ тире перед годом *)
year := CONCAT(tire, year_not_tire);				(* Объединяем тире и год *)

conc1 := CONCAT(day, month);					(* Объединяем день и месяц *)
conc2 := CONCAT(conc1, year);					(* Объединяем день, месяц и год *)

stDate := conc2;								(* Текущая дата *)
stTime := MID(output_time, 11, 5);				(* Текущее время *)
stTime_graphic := LEFT (stTime, 5);				(* Отделяю секунды, оставив часы и минуты *)

stDate_Alarm := conc2;							(* Текущая дата для Аварий *)
stTime_Alarm := MID(output_time, 11, 5);			(* Текущее время для Аварий *)


(*------------- Запись данных в одну переменную ---------------*)
razdelitel := ' | ';										(* Задаем разделитель для удодного отображения сообщения *)
stDate_r := CONCAT(stDate_Alarm, razdelitel);		(* Объединяем дату и разделитель *)
stTime_r := CONCAT(stTime_Alarm, razdelitel);		(* Объединяем время и разделитель *)

stDate_and_Time := CONCAT(stDate_Alarm, stTime_Alarm );			(* Объединяем дату и время в уже удобной для нас форме *)



(*------------- 	ОПРЕДЕЛЕНИЕ ДНЯ НЕДЕЛИ -------------*)

NumOfDay := DATE_TO_DWORD(input_date) / 86400;
NumOfDay := NumOfDay + 3;
DAY_OF_WEEK := DWORD_TO_UINT(NumOfDay MOD 7);



(* Тестовая часть для проверки всех дней недели *)

IF DAY_OF_WEEK = 0 THEN
	Day_of_Today := ' Пн ';
ELSIF DAY_OF_WEEK = 1 THEN
	Day_of_Today := ' Вт ';
ELSIF DAY_OF_WEEK = 2 THEN
	Day_of_Today := ' Ср ';
ELSIF DAY_OF_WEEK = 3 THEN
	Day_of_Today := ' Чт ';
ELSIF DAY_OF_WEEK = 4 THEN
	Day_of_Today := ' Пт ';
ELSIF DAY_OF_WEEK = 5 THEN
	Day_of_Today := ' Сб ';
ELSIF DAY_OF_WEEK = 6 THEN
	Day_of_Today := ' Вс ';
END_IF
END_PROGRAM

(* POU LAMPS, ST *)
PROGRAM LAMPS
VAR
	LAMP_HL1					: STRING	:=' ';
	tmOnPoloska				: TON;
	tmOffPoloska				: TON;
	tm_AlarmPoloska			: TP;
	AlarmPoloska				: BOOL;
	AlarmPoloska_invisible		: BOOL;
	buttonFillColorAlarm			: DWORD;
	buttonTextFillColorAlarm		: DWORD;
END_VAR
(*---------------- АВАРИЯ ВХОДНОГО НАПРЯЖЕНИЯ --------*)

IF K152_1SHA1_QF1 THEN
	LAMP_HL1:=' Сеть ';
	K152_1SHA1_HL1 := TRUE;
ELSE
	K152_1SHA1_HL1 := FALSE;
	LAMP_HL1:=' ';
END_IF

(*---------------- АВАРИЙНАЯ ПОЛОСКА--------------------------------------------*)
AlarmPoloska_invisible := NOT(AlarmPoloska);
IF i <> 0 THEN
	tmOnPoloska ( IN := TRUE , PT := T#400ms );
ELSE
	AlarmPoloska := FALSE;
	tmOnPoloska ( IN := FALSE , PT := T#400ms );
	tmOffPoloska ( IN:= FALSE , PT:=T#400ms );
	buttonFillColorAlarm := 16#000000;
	buttonTextFillColorAlarm := 16#000000;
END_IF

IF tmOnPoloska.Q THEN
	AlarmPoloska := TRUE;
	tmOnPoloska ( IN := FALSE , PT := T#400ms );
	tmOffPoloska ( IN:= TRUE , PT:=T#400ms );
	buttonFillColorAlarm := 16#0000FF;
	buttonTextFillColorAlarm := 16#0000FF;
END_IF

IF tmOffPoloska.Q THEN
	AlarmPoloska := FALSE;
	tmOnPoloska ( IN := TRUE , PT := T#400ms );
	tmOffPoloska ( IN:= FALSE , PT:=T#400ms );
	buttonFillColorAlarm := 16#000000;
	buttonTextFillColorAlarm := 16#000000;
END_IF
END_PROGRAM

(* POU VHOD, ST *)
PROGRAM VHOD
VAR
	Password						: STRING := '';
	bMAIN_PAGE					: BOOL;
	FAIL_PASS_TEXT				: STRING := 'НЕВЕРНЫЙ ПАРОЛЬ';
	FAIL_PASS						: BOOL;
	User							: STRING := 'Авторизация';
	Vihod							: BOOL;
	bVihod							: BOOL;
	TECHNIK						: BOOL;
	bOK							: BOOL;
	bAUTORIZATION				: BOOL;
	AUTORIZATION_INVISIBLE		: BOOL := TRUE;
	rt_AVTORIZATION				: R_TRIG;
	INVISIBLE_ELEMENT			: BOOL;
END_VAR
IF Password='1575' THEN
	bOK:=FALSE;
	bMAIN_PAGE:=FALSE;
	User:='Инженер';
	FAIL_PASS:=TRUE;
	INVISIBLE_ELEMENT:=FALSE;
ELSIF Password='6666' THEN
	FAIL_PASS:=TRUE;
	User:='Техник';
	TECHNIK:=TRUE;
	bOK:=FALSE;
	INVISIBLE_ELEMENT:=TRUE;
ELSE
	FAIL_PASS:=FALSE;
	bMAIN_PAGE:=FALSE;
	User:='Авторизация';
	bOK:=TRUE;
END_IF

rt_AVTORIZATION (CLK:=bAUTORIZATION);

IF rt_AVTORIZATION.Q THEN
	AUTORIZATION_INVISIBLE:=FALSE;
END_IF

IF Password=''THEN
	FAIL_PASS:=TRUE;
END_IF

IF bVihod THEN
	AUTORIZATION_INVISIBLE:=TRUE;
	bVihod:=FALSE;
	Password:='';
	User:='Авторизация';
END_IF
END_PROGRAM

(* POU SCHAO1, ST *)
PROGRAM SCHAO1
VAR
	rt_K152_1SHA1_SCHAO1_LIGHT_GR5_ON				: R_TRIG;		(* Кнопка включения группы освещения. гр.5 *)
	rt_K152_1SHA1_SCHAO1_LIGHT_GR5_OFF				: R_TRIG;		(* Кнопка выключения группы освещения. гр.5 *)
END_VAR
(* Столбец 1 *)
masTABLE_SCHAO1[1].s1Positioin := ' Наличие напряжения на вводе ';
masTABLE_SCHAO1[2].s1Positioin := ' Автоматический выключатель QF1 ';
masTABLE_SCHAO1[3].s1Positioin := ' Автоматический выключатель QF2 ';
masTABLE_SCHAO1[4].s1Positioin := ' Автоматический выключатель QF3 ';
masTABLE_SCHAO1[5].s1Positioin := ' Автоматический выключатель QF4 ';
masTABLE_SCHAO1[6].s1Positioin := ' Автоматический выключатель QF5 ';
masTABLE_SCHAO1[7].s1Positioin := ' Автоматический выключатель QF6 ';
masTABLE_SCHAO1[8].s1Positioin := ' Автоматический выключатель QF7 ';
masTABLE_SCHAO1[9].s1Positioin := ' Положение магнитного пускателя гр.5 ';
masTABLE_SCHAO1[10].s1Positioin := ' Положение переключателя в режиме Авт. гр.5 ';
masTABLE_SCHAO1[11].s1Positioin := ' Положение переключателя в режиме Руч. гр.5 ';

(* Столбец 2 *)
masTABLE_SCHAO1[1].s2Value_X := st_SCHAO1_POWER;
masTABLE_SCHAO1[2].s2Value_X := st_SCHAO1_QF1;
masTABLE_SCHAO1[3].s2Value_X := st_SCHAO1_QF2;
masTABLE_SCHAO1[4].s2Value_X := st_SCHAO1_QF3;
masTABLE_SCHAO1[5].s2Value_X := st_SCHAO1_QF4;
masTABLE_SCHAO1[6].s2Value_X := st_SCHAO1_QF5;
masTABLE_SCHAO1[7].s2Value_X := st_SCHAO1_QF6;
masTABLE_SCHAO1[8].s2Value_X := st_SCHAO1_QF7;
masTABLE_SCHAO1[9].s2Value_X := st_SCHAO1_KM_GR5;
masTABLE_SCHAO1[10].s2Value_X := st_SCHAO1_SA_AVT_GR5;
masTABLE_SCHAO1[11].s2Value_X := st_SCHAO1_SA_RUCH_GR5;


(* Отображение состояния *)
IF K152_1SHA1_SCHAO1_POWER THEN
	st_SCHAO1_POWER := ' Включено ';
	masTABLE_SCHAO1[1].dwFillColorAlarm := 16#00FF00;
ELSE
	st_SCHAO1_POWER := ' Выключено ';
	masTABLE_SCHAO1[1].dwFillColorAlarm := 16#FFFFEF;
END_IF

IF K152_1SHA1_SCHAO1_QF1 THEN
	st_SCHAO1_QF1 := ' Включено ';
	masTABLE_SCHAO1[2].dwFillColorAlarm := 16#00FF00;
ELSE
	st_SCHAO1_QF1 := ' Выключено ';
	masTABLE_SCHAO1[2].dwFillColorAlarm := 16#FFFFEF;
END_IF

IF K152_1SHA1_SCHAO1_QF2 THEN
	st_SCHAO1_QF2 := ' Включено ';
	masTABLE_SCHAO1[3].dwFillColorAlarm := 16#00FF00;
ELSE
	st_SCHAO1_QF2 := ' Выключено ';
	masTABLE_SCHAO1[3].dwFillColorAlarm := 16#FFFFEF;
END_IF

IF K152_1SHA1_SCHAO1_QF3 THEN
	st_SCHAO1_QF3 := ' Включено ';
	masTABLE_SCHAO1[4].dwFillColorAlarm := 16#00FF00;
ELSE
	st_SCHAO1_QF3 := ' Выключено ';
	masTABLE_SCHAO1[4].dwFillColorAlarm := 16#FFFFEF;
END_IF

IF K152_1SHA1_SCHAO1_QF4 THEN
	st_SCHAO1_QF4 := ' Включено ';
	masTABLE_SCHAO1[5].dwFillColorAlarm := 16#00FF00;
ELSE
	st_SCHAO1_QF4 := ' Выключено ';
	masTABLE_SCHAO1[5].dwFillColorAlarm := 16#FFFFEF;
END_IF

IF K152_1SHA1_SCHAO1_QF5 THEN
	st_SCHAO1_QF5 := ' Включено ';
	masTABLE_SCHAO1[6].dwFillColorAlarm := 16#00FF00;
ELSE
	st_SCHAO1_QF5 := ' Выключено ';
	masTABLE_SCHAO1[6].dwFillColorAlarm := 16#FFFFEF;
END_IF

IF K152_1SHA1_SCHAO1_QF6 THEN
	st_SCHAO1_QF6 := ' Включено ';
	masTABLE_SCHAO1[7].dwFillColorAlarm := 16#00FF00;
ELSE
	st_SCHAO1_QF6 := ' Выключено ';
	masTABLE_SCHAO1[7].dwFillColorAlarm := 16#FFFFEF;
END_IF

IF K152_1SHA1_SCHAO1_QF7 THEN
	st_SCHAO1_QF7 := ' Включено ';
	masTABLE_SCHAO1[8].dwFillColorAlarm := 16#00FF00;
ELSE
	st_SCHAO1_QF7 := ' Выключено ';
	masTABLE_SCHAO1[8].dwFillColorAlarm := 16#FFFFEF;
END_IF

IF K152_1SHA1_SCHAO1_KM_GR5 THEN
	st_SCHAO1_KM_GR5 := ' Включено ';
	masTABLE_SCHAO1[9].dwFillColorAlarm := 16#00FF00;
ELSE
	st_SCHAO1_KM_GR5 := ' Выключено ';
	masTABLE_SCHAO1[9].dwFillColorAlarm := 16#FFFFEF;
END_IF

IF K152_1SHA1_SCHAO1_SA_AVT_GR5 THEN
	st_SCHAO1_SA_AVT_GR5 := ' Включено ';
	masTABLE_SCHAO1[10].dwFillColorAlarm := 16#00FF00;
ELSE
	st_SCHAO1_SA_AVT_GR5 := ' Выключено ';
	masTABLE_SCHAO1[10].dwFillColorAlarm := 16#FFFFEF;
END_IF

IF K152_1SHA1_SCHAO1_SA_RUCH_GR5 THEN
	st_SCHAO1_SA_RUCH_GR5 := ' Включено ';
	masTABLE_SCHAO1[11].dwFillColorAlarm := 16#00FF00;
ELSE
	st_SCHAO1_SA_RUCH_GR5 := ' Выключено ';
	masTABLE_SCHAO1[11].dwFillColorAlarm := 16#FFFFEF;
END_IF


(* Управление *)
rt_K152_1SHA1_SCHAO1_LIGHT_GR5_ON		( CLK := bK152_1SHA1_SCHAO1_LIGHT_GR5_ON );
rt_K152_1SHA1_SCHAO1_LIGHT_GR5_OFF		( CLK := bK152_1SHA1_SCHAO1_LIGHT_GR5_OFF );

(* Управление освещением гр.5 *)
IF rt_K152_1SHA1_SCHAO1_LIGHT_GR5_ON.Q THEN
	bK152_1SHA1_SCHAO1_LIGHT_GR5_OFF := FALSE;
	K152_1SHA1_SCHAO1_LIGHT_GR5 := TRUE;
ELSIF rt_K152_1SHA1_SCHAO1_LIGHT_GR5_OFF.Q THEN
	bK152_1SHA1_SCHAO1_LIGHT_GR5_ON := FALSE;
	K152_1SHA1_SCHAO1_LIGHT_GR5 := FALSE;
END_IF
END_PROGRAM

(* POU SCHAO2, ST *)
PROGRAM SCHAO2
VAR
	rt_K152_1SHA1_SCHAO2_LIGHT_GR5_ON				: R_TRIG;		(* Кнопка включения группы освещения. гр.5 *)
	rt_K152_1SHA1_SCHAO2_LIGHT_GR5_OFF				: R_TRIG;		(* Кнопка выключения группы освещения. гр.5 *)
END_VAR
(* Столбец 1 *)
masTABLE_SCHAO2[1].s1Positioin := ' Наличие напряжения на вводе ';
masTABLE_SCHAO2[2].s1Positioin := ' Автоматический выключатель QF1 ';
masTABLE_SCHAO2[3].s1Positioin := ' Автоматический выключатель QF2 ';
masTABLE_SCHAO2[4].s1Positioin := ' Автоматический выключатель QF3 ';
masTABLE_SCHAO2[5].s1Positioin := ' Автоматический выключатель QF4 ';
masTABLE_SCHAO2[6].s1Positioin := ' Автоматический выключатель QF5 ';
masTABLE_SCHAO2[7].s1Positioin := ' Автоматический выключатель QF6 ';
masTABLE_SCHAO2[8].s1Positioin := ' Автоматический выключатель QF7 ';
masTABLE_SCHAO2[9].s1Positioin := ' Автоматический выключатель QF8 ';
masTABLE_SCHAO2[10].s1Positioin := ' Автоматический выключатель QF9 ';
masTABLE_SCHAO2[11].s1Positioin := ' Положение магнитного пускателя гр.5 ';
masTABLE_SCHAO2[12].s1Positioin := ' Положение переключателя в режиме Авт. гр.5 ';
masTABLE_SCHAO2[13].s1Positioin := ' Положение переключателя в режиме Руч. гр.5 ';

(* Столбец 2 *)
masTABLE_SCHAO2[1].s2Value_X := st_SCHAO2_POWER;
masTABLE_SCHAO2[2].s2Value_X := st_SCHAO2_QF1;
masTABLE_SCHAO2[3].s2Value_X := st_SCHAO2_QF2;
masTABLE_SCHAO2[4].s2Value_X := st_SCHAO2_QF3;
masTABLE_SCHAO2[5].s2Value_X := st_SCHAO2_QF4;
masTABLE_SCHAO2[6].s2Value_X := st_SCHAO2_QF5;
masTABLE_SCHAO2[7].s2Value_X := st_SCHAO2_QF6;
masTABLE_SCHAO2[8].s2Value_X := st_SCHAO2_QF7;
masTABLE_SCHAO2[9].s2Value_X := st_SCHAO2_QF8;
masTABLE_SCHAO2[10].s2Value_X := st_SCHAO2_QF9;
masTABLE_SCHAO2[11].s2Value_X := st_SCHAO2_KM_GR5;
masTABLE_SCHAO2[12].s2Value_X := st_SCHAO2_SA_AVT_GR5;
masTABLE_SCHAO2[13].s2Value_X := st_SCHAO2_SA_RUCH_GR5;

(* Отображение состояния *)
IF K152_1SHA1_SCHAO2_POWER THEN
	st_SCHAO2_POWER := ' Включено ';
	masTABLE_SCHAO2[1].dwFillColorAlarm := 16#00FF00;
ELSE
	st_SCHAO2_POWER := ' Выключено ';
	masTABLE_SCHAO2[1].dwFillColorAlarm := 16#FFFFEF;
END_IF

IF K152_1SHA1_SCHAO2_QF1 THEN
	st_SCHAO2_QF1 := ' Включено ';
	masTABLE_SCHAO2[2].dwFillColorAlarm := 16#00FF00;
ELSE
	st_SCHAO2_QF1 := ' Выключено ';
	masTABLE_SCHAO2[2].dwFillColorAlarm := 16#FFFFEF;
END_IF

IF K152_1SHA1_SCHAO2_QF2 THEN
	st_SCHAO2_QF2 := ' Включено ';
	masTABLE_SCHAO2[3].dwFillColorAlarm := 16#00FF00;
ELSE
	st_SCHAO2_QF2 := ' Выключено ';
	masTABLE_SCHAO2[3].dwFillColorAlarm := 16#FFFFEF;
END_IF

IF K152_1SHA1_SCHAO2_QF3 THEN
	st_SCHAO2_QF3 := ' Включено ';
	masTABLE_SCHAO2[4].dwFillColorAlarm := 16#00FF00;
ELSE
	st_SCHAO2_QF3 := ' Выключено ';
	masTABLE_SCHAO2[4].dwFillColorAlarm := 16#FFFFEF;
END_IF

IF K152_1SHA1_SCHAO2_QF4 THEN
	st_SCHAO2_QF4 := ' Включено ';
	masTABLE_SCHAO2[5].dwFillColorAlarm := 16#00FF00;
ELSE
	st_SCHAO2_QF4 := ' Выключено ';
	masTABLE_SCHAO2[5].dwFillColorAlarm := 16#FFFFEF;
END_IF

IF K152_1SHA1_SCHAO2_QF5 THEN
	st_SCHAO2_QF5 := ' Включено ';
	masTABLE_SCHAO2[6].dwFillColorAlarm := 16#00FF00;
ELSE
	st_SCHAO2_QF5 := ' Выключено ';
	masTABLE_SCHAO2[6].dwFillColorAlarm := 16#FFFFEF;
END_IF

IF K152_1SHA1_SCHAO2_QF6 THEN
	st_SCHAO2_QF6 := ' Включено ';
	masTABLE_SCHAO2[7].dwFillColorAlarm := 16#00FF00;
ELSE
	st_SCHAO2_QF6 := ' Выключено ';
	masTABLE_SCHAO2[7].dwFillColorAlarm := 16#FFFFEF;
END_IF

IF K152_1SHA1_SCHAO2_QF7 THEN
	st_SCHAO2_QF7 := ' Включено ';
	masTABLE_SCHAO2[8].dwFillColorAlarm := 16#00FF00;
ELSE
	st_SCHAO2_QF7 := ' Выключено ';
	masTABLE_SCHAO2[8].dwFillColorAlarm := 16#FFFFEF;
END_IF

IF K152_1SHA1_SCHAO2_QF8 THEN
	st_SCHAO2_QF8 := ' Включено ';
	masTABLE_SCHAO2[9].dwFillColorAlarm := 16#00FF00;
ELSE
	st_SCHAO2_QF8 := ' Выключено ';
	masTABLE_SCHAO2[9].dwFillColorAlarm := 16#FFFFEF;
END_IF

IF K152_1SHA1_SCHAO2_QF9 THEN
	st_SCHAO2_QF9 := ' Включено ';
	masTABLE_SCHAO2[10].dwFillColorAlarm := 16#00FF00;
ELSE
	st_SCHAO2_QF9 := ' Выключено ';
	masTABLE_SCHAO2[10].dwFillColorAlarm := 16#FFFFEF;
END_IF

IF K152_1SHA1_SCHAO2_KM_GR5 THEN
	st_SCHAO2_KM_GR5 := ' Включено ';
	masTABLE_SCHAO2[11].dwFillColorAlarm := 16#00FF00;
ELSE
	st_SCHAO2_KM_GR5 := ' Выключено ';
	masTABLE_SCHAO2[11].dwFillColorAlarm := 16#FFFFEF;
END_IF

IF K152_1SHA1_SCHAO2_SA_AVT_GR5 THEN
	st_SCHAO2_SA_AVT_GR5 := ' Включено ';
	masTABLE_SCHAO2[12].dwFillColorAlarm := 16#00FF00;
ELSE
	st_SCHAO2_SA_AVT_GR5 := ' Выключено ';
	masTABLE_SCHAO2[12].dwFillColorAlarm := 16#FFFFEF;
END_IF

IF K152_1SHA1_SCHAO2_SA_RUCH_GR5 THEN
	st_SCHAO2_SA_RUCH_GR5 := ' Включено ';
	masTABLE_SCHAO2[13].dwFillColorAlarm := 16#00FF00;
ELSE
	st_SCHAO2_SA_RUCH_GR5 := ' Выключено ';
	masTABLE_SCHAO2[13].dwFillColorAlarm := 16#FFFFEF;
END_IF


(* Управление *)
rt_K152_1SHA1_SCHAO2_LIGHT_GR5_ON		( CLK := bK152_1SHA1_SCHAO2_LIGHT_GR5_ON );
rt_K152_1SHA1_SCHAO2_LIGHT_GR5_OFF		( CLK := bK152_1SHA1_SCHAO2_LIGHT_GR5_OFF );

(* Управление освещением гр.5 *)
IF rt_K152_1SHA1_SCHAO2_LIGHT_GR5_ON.Q THEN
	bK152_1SHA1_SCHAO2_LIGHT_GR5_OFF := FALSE;
	K152_1SHA1_SCHAO2_LIGHT_GR5 := TRUE;
ELSIF rt_K152_1SHA1_SCHAO2_LIGHT_GR5_OFF.Q THEN
	bK152_1SHA1_SCHAO2_LIGHT_GR5_ON := FALSE;
	K152_1SHA1_SCHAO2_LIGHT_GR5 := FALSE;
END_IF
END_PROGRAM

(* POU SCHO1, ST *)
PROGRAM SCHO1
VAR
	rt_K152_1SHA1_SCHO1_LIGHT_GR1_ON		: R_TRIG;		(* Кнопка включения группы освещения. гр.1 *)
	rt_K152_1SHA1_SCHO1_LIGHT_GR1_OFF		: R_TRIG;		(* Кнопка выключения группы освещения. гр.1 *)
	rt_K152_1SHA1_SCHO1_LIGHT_GR2_ON		: R_TRIG;		(* Кнопка включения группы освещения. гр.2 *)
	rt_K152_1SHA1_SCHO1_LIGHT_GR2_OFF		: R_TRIG;		(* Кнопка выключения группы освещения. гр.2 *)
END_VAR
(* Столбец 1 *)
masTABLE_SCHO1[1].s1Positioin := ' Автоматический выключатель QF1 ';
masTABLE_SCHO1[2].s1Positioin := ' Автоматический выключатель QF2 ';
masTABLE_SCHO1[3].s1Positioin := ' Положение магнитного пускателя гр.1 ';
masTABLE_SCHO1[4].s1Positioin := ' Положение магнитного пускателя гр.2 ';
masTABLE_SCHO1[5].s1Positioin := ' Положение переключателя в режиме Авт. гр.1 ';
masTABLE_SCHO1[6].s1Positioin := ' Положение переключателя в режиме Авт. гр.2 ';
masTABLE_SCHO1[7].s1Positioin := ' Положение переключателя в режиме Руч. гр.1 ';
masTABLE_SCHO1[8].s1Positioin := ' Положение переключателя в режиме Руч. гр.2 ';

(* Столбец 2 *)
masTABLE_SCHO1[1].s2Value_X := st_SCHO1_QF1;
masTABLE_SCHO1[2].s2Value_X := st_SCHO1_QF2;
masTABLE_SCHO1[3].s2Value_X := st_SCHO1_KM_GR1;
masTABLE_SCHO1[4].s2Value_X := st_SCHO1_KM_GR2;
masTABLE_SCHO1[5].s2Value_X := st_SCHO1_SA_AVT_GR1;
masTABLE_SCHO1[6].s2Value_X := st_SCHO1_SA_AVT_GR2;
masTABLE_SCHO1[7].s2Value_X := st_SCHO1_SA_RUCH_GR1;
masTABLE_SCHO1[8].s2Value_X := st_SCHO1_SA_RUCH_GR2;

(* Отображение состояния *)
IF K152_1SHA1_SCHO1_QF1 THEN
	st_SCHO1_QF1 := ' Включено ';
	masTABLE_SCHO1[1].dwFillColorAlarm := 16#00FF00;
ELSE
	st_SCHO1_QF1 := ' Выключено ';
	masTABLE_SCHO1[1].dwFillColorAlarm := 16#FFFFEF;
END_IF

IF K152_1SHA1_SCHO1_QF2 THEN
	st_SCHO1_QF2 := ' Включено ';
	masTABLE_SCHO1[2].dwFillColorAlarm := 16#00FF00;
ELSE
	st_SCHO1_QF2 := ' Выключено ';
	masTABLE_SCHO1[2].dwFillColorAlarm := 16#FFFFEF;
END_IF

IF K152_1SHA1_SCHO1_KM_GR1 THEN
	st_SCHO1_KM_GR1 := ' Включено ';
	masTABLE_SCHO1[3].dwFillColorAlarm := 16#00FF00;
ELSE
	st_SCHO1_KM_GR1 := ' Выключено ';
	masTABLE_SCHO1[3].dwFillColorAlarm := 16#FFFFEF;
END_IF

IF K152_1SHA1_SCHO1_KM_GR2 THEN
	st_SCHO1_KM_GR2 := ' Включено ';
	masTABLE_SCHO1[4].dwFillColorAlarm := 16#00FF00;
ELSE
	st_SCHO1_KM_GR2 := ' Выключено ';
	masTABLE_SCHO1[4].dwFillColorAlarm := 16#FFFFEF;
END_IF

IF K152_1SHA1_SCHO1_SA_AVT_GR1 THEN
	st_SCHO1_SA_AVT_GR1 := ' Включено ';
	masTABLE_SCHO1[5].dwFillColorAlarm := 16#00FF00;
ELSE
	st_SCHO1_SA_AVT_GR1 := ' Выключено ';
	masTABLE_SCHO1[5].dwFillColorAlarm := 16#FFFFEF;
END_IF

IF K152_1SHA1_SCHO1_SA_AVT_GR2 THEN
	st_SCHO1_SA_AVT_GR2 := ' Включено ';
	masTABLE_SCHO1[6].dwFillColorAlarm := 16#00FF00;
ELSE
	st_SCHO1_SA_AVT_GR2 := ' Выключено ';
	masTABLE_SCHO1[6].dwFillColorAlarm := 16#FFFFEF;
END_IF

IF K152_1SHA1_SCHO1_SA_RUCH_GR1 THEN
	st_SCHO1_SA_RUCH_GR1 := ' Включено ';
	masTABLE_SCHO1[7].dwFillColorAlarm := 16#00FF00;
ELSE
	st_SCHO1_SA_RUCH_GR1 := ' Выключено ';
	masTABLE_SCHO1[7].dwFillColorAlarm := 16#FFFFEF;
END_IF

IF K152_1SHA1_SCHO1_SA_RUCH_GR2 THEN
	st_SCHO1_SA_RUCH_GR2 := ' Включено ';
	masTABLE_SCHO1[8].dwFillColorAlarm := 16#00FF00;
ELSE
	st_SCHO1_SA_RUCH_GR2 := ' Выключено ';
	masTABLE_SCHO1[8].dwFillColorAlarm := 16#FFFFEF;
END_IF

(* Управление *)
rt_K152_1SHA1_SCHO1_LIGHT_GR1_ON		( CLK := bK152_1SHA1_SCHO1_LIGHT_GR1_ON );
rt_K152_1SHA1_SCHO1_LIGHT_GR1_OFF		( CLK := bK152_1SHA1_SCHO1_LIGHT_GR1_OFF );
rt_K152_1SHA1_SCHO1_LIGHT_GR2_ON		( CLK := bK152_1SHA1_SCHO1_LIGHT_GR2_ON );
rt_K152_1SHA1_SCHO1_LIGHT_GR2_OFF		( CLK := bK152_1SHA1_SCHO1_LIGHT_GR2_OFF );

(* Управление освещением гр.1 *)
IF rt_K152_1SHA1_SCHO1_LIGHT_GR1_ON.Q THEN
	bK152_1SHA1_SCHO1_LIGHT_GR1_OFF := FALSE;
	K152_1SHA1_SCHO1_LIGHT_GR1 := TRUE;
ELSIF rt_K152_1SHA1_SCHO1_LIGHT_GR1_OFF.Q THEN
	bK152_1SHA1_SCHO1_LIGHT_GR1_ON := FALSE;
	K152_1SHA1_SCHO1_LIGHT_GR1 := FALSE;
END_IF
(* Управление освещением гр.2 *)
IF rt_K152_1SHA1_SCHO1_LIGHT_GR2_ON.Q THEN
	bK152_1SHA1_SCHO1_LIGHT_GR2_OFF := FALSE;
	K152_1SHA1_SCHO1_LIGHT_GR2 := TRUE;
ELSIF rt_K152_1SHA1_SCHO1_LIGHT_GR2_OFF.Q THEN
	bK152_1SHA1_SCHO1_LIGHT_GR2_ON := FALSE;
	K152_1SHA1_SCHO1_LIGHT_GR2 := FALSE;
END_IF
END_PROGRAM

(* POU SCHO2, ST *)
PROGRAM SCHO2
VAR
	rt_bK152_1SHA1_SCHO2_LIGHT_GR1_ON		: R_TRIG;		(* Кнопка включения группы освещения. гр.1 *)
	rt_bK152_1SHA1_SCHO2_LIGHT_GR2_ON		: R_TRIG;		(* Кнопка включения группы освещения. гр.2 *)
	rt_bK152_1SHA1_SCHO2_LIGHT_GR3_ON		: R_TRIG;		(* Кнопка включения группы освещения. гр.3 *)
	rt_bK152_1SHA1_SCHO2_LIGHT_GR4_ON		: R_TRIG;		(* Кнопка включения группы освещения. гр.4 *)
	rt_bK152_1SHA1_SCHO2_LIGHT_GR5_ON		: R_TRIG;		(* Кнопка включения группы освещения. гр.5 *)
	rt_bK152_1SHA1_SCHO2_LIGHT_GR9_ON		: R_TRIG;		(* Кнопка включения группы освещения. гр.9 *)

	rt_bK152_1SHA1_SCHO2_LIGHT_GR1_OFF		: R_TRIG;		(* Кнопка выключения группы освещения. гр.1 *)
	rt_bK152_1SHA1_SCHO2_LIGHT_GR2_OFF		: R_TRIG;		(* Кнопка выключения группы освещения. гр.2 *)
	rt_bK152_1SHA1_SCHO2_LIGHT_GR3_OFF		: R_TRIG;		(* Кнопка выключения группы освещения. гр.3 *)
	rt_bK152_1SHA1_SCHO2_LIGHT_GR4_OFF		: R_TRIG;		(* Кнопка выключения группы освещения. гр.4 *)
	rt_bK152_1SHA1_SCHO2_LIGHT_GR5_OFF		: R_TRIG;		(* Кнопка выключения группы освещения. гр.5 *)
	rt_bK152_1SHA1_SCHO2_LIGHT_GR9_OFF		: R_TRIG;		(* Кнопка выключения группы освещения. гр.9 *)
END_VAR
(* ОСВЕЩЕНИЕ ГРУППА 1 *)
(* Столбец 1 *)
masTABLE_SCHO2_1[1].Position := ' Автоматический выключатель QF1 ';
masTABLE_SCHO2_1[2].Position := ' Положение магнитного пускателя ';
masTABLE_SCHO2_1[3].Position := ' Положение переключателя в режиме АВТ. ';
masTABLE_SCHO2_1[4].Position := ' Положение переключателя в режиме РУЧ. ';
(* Столбец 2 *)
IF K152_1SHA1_SCHO2_QF1 THEN
	masTABLE_SCHO2_1[1].On_Off := ' Включено ';
	masTABLE_SCHO2_1[1].ON := TRUE;
ELSE
	masTABLE_SCHO2_1[1].On_Off := ' Выключено ';
	masTABLE_SCHO2_1[1].ON := FALSE;
END_IF

IF K152_1SHA1_SCHO2_KM_GR1 THEN
	st_SCHO2_KM_GR1 := ' Включено ';
	masTABLE_SCHO2_1[2].dwFillColorAlarm := 16#00FF00;
ELSE
	st_SCHO2_KM_GR1 := ' Выключено ';
	masTABLE_SCHO2_1[2].dwFillColorAlarm := 16#FFFFEF;
END_IF

IF K152_1SHA1_SCHO2_SA_AVT_GR1 THEN
	st_SCHO2_SA_AVT_GR1 := ' Включено ';
	masTABLE_SCHO2_1[3].dwFillColorAlarm := 16#00FF00;
ELSE
	st_SCHO2_SA_AVT_GR1 := ' Выключено ';
	masTABLE_SCHO2_1[3].dwFillColorAlarm := 16#FFFFEF;
END_IF

IF K152_1SHA1_SCHO2_SA_RUCH_GR1 THEN
	st_SCHO2_SA_RUCH_GR1 := ' Включено ';
	masTABLE_SCHO2_1[4].dwFillColorAlarm := 16#00FF00;
ELSE
	st_SCHO2_SA_RUCH_GR1 := ' Выключено ';
	masTABLE_SCHO2_1[4].dwFillColorAlarm := 16#FFFFEF;
END_IF

(* Управление освещением гр.1 *)
rt_bK152_1SHA1_SCHO2_LIGHT_GR1_ON		( CLK := bK152_1SHA1_SCHO2_LIGHT_GR1_ON );
rt_bK152_1SHA1_SCHO2_LIGHT_GR1_OFF		( CLK := bK152_1SHA1_SCHO2_LIGHT_GR1_OFF );

IF rt_bK152_1SHA1_SCHO2_LIGHT_GR1_ON.Q THEN
	bK152_1SHA1_SCHO2_LIGHT_GR1_OFF := FALSE;
	K152_1SHA1_SCHO2_LIGHT_GR1 := TRUE;
ELSIF rt_bK152_1SHA1_SCHO2_LIGHT_GR1_OFF.Q THEN
	bK152_1SHA1_SCHO2_LIGHT_GR1_ON := FALSE;
	K152_1SHA1_SCHO2_LIGHT_GR1 := FALSE;
END_IF


(* ОСВЕЩЕНИЕ ГРУППА 2 *)
(* Столбец 1 *)
masTABLE_SCHO2_2[1].s1Positioin := ' Автоматический выключатель QF2 ';
masTABLE_SCHO2_2[2].s1Positioin := ' Положение магнитного пускателя ';
masTABLE_SCHO2_2[3].s1Positioin := ' Положение переключателя в режиме АВТ. ';
masTABLE_SCHO2_2[4].s1Positioin := ' Положение переключателя в режиме РУЧ. ';
(* Столбец 2 *)
masTABLE_SCHO2_2[1].s2Value_X := st_SCHO2_QF2;
masTABLE_SCHO2_2[2].s2Value_X := st_SCHO2_KM_GR2;
masTABLE_SCHO2_2[3].s2Value_X := st_SCHO2_SA_AVT_GR2;
masTABLE_SCHO2_2[4].s2Value_X := st_SCHO2_SA_RUCH_GR2;
(* Отображение состояния *)
IF K152_1SHA1_SCHO2_QF2 THEN
	st_SCHO2_QF2 := ' Включено ';
	masTABLE_SCHO2_2[1].dwFillColorAlarm := 16#00FF00;
ELSE
	st_SCHO2_QF2 := ' Выключено ';
	masTABLE_SCHO2_2[1].dwFillColorAlarm := 16#FFFFEF;
END_IF

IF K152_1SHA1_SCHO2_KM_GR2 THEN
	st_SCHO2_KM_GR2 := ' Включено ';
	masTABLE_SCHO2_2[2].dwFillColorAlarm := 16#00FF00;
ELSE
	st_SCHO2_KM_GR2 := ' Выключено ';
	masTABLE_SCHO2_2[2].dwFillColorAlarm := 16#FFFFEF;
END_IF

IF K152_1SHA1_SCHO2_SA_AVT_GR2 THEN
	st_SCHO2_SA_AVT_GR2 := ' Включено ';
	masTABLE_SCHO2_2[3].dwFillColorAlarm := 16#00FF00;
ELSE
	st_SCHO2_SA_AVT_GR2 := ' Выключено ';
	masTABLE_SCHO2_2[3].dwFillColorAlarm := 16#FFFFEF;
END_IF

IF K152_1SHA1_SCHO2_SA_RUCH_GR2 THEN
	st_SCHO2_SA_RUCH_GR2 := ' Включено ';
	masTABLE_SCHO2_2[4].dwFillColorAlarm := 16#00FF00;
ELSE
	st_SCHO2_SA_RUCH_GR2 := ' Выключено ';
	masTABLE_SCHO2_2[4].dwFillColorAlarm := 16#FFFFEF;
END_IF

(* Управление освещением гр.2 *)
rt_bK152_1SHA1_SCHO2_LIGHT_GR2_ON		( CLK := bK152_1SHA1_SCHO2_LIGHT_GR2_ON );
rt_bK152_1SHA1_SCHO2_LIGHT_GR2_OFF		( CLK := bK152_1SHA1_SCHO2_LIGHT_GR2_OFF );

IF rt_bK152_1SHA1_SCHO2_LIGHT_GR2_ON.Q THEN
	bK152_1SHA1_SCHO2_LIGHT_GR2_OFF := FALSE;
	K152_1SHA1_SCHO2_LIGHT_GR2 := TRUE;
ELSIF rt_bK152_1SHA1_SCHO2_LIGHT_GR2_OFF.Q THEN
	bK152_1SHA1_SCHO2_LIGHT_GR2_ON := FALSE;
	K152_1SHA1_SCHO2_LIGHT_GR2 := FALSE;
END_IF


(* ОСВЕЩЕНИЕ ГРУППА 3 *)
(* Столбец 1 *)
masTABLE_SCHO2_3[1].s1Positioin := ' Автоматический выключатель QF3 ';
masTABLE_SCHO2_3[2].s1Positioin := ' Положение магнитного пускателя ';
masTABLE_SCHO2_3[3].s1Positioin := ' Положение переключателя в режиме АВТ. ';
masTABLE_SCHO2_3[4].s1Positioin := ' Положение переключателя в режиме РУЧ. ';
(* Столбец 2 *)
masTABLE_SCHO2_3[1].s2Value_X := st_SCHO2_QF3;
masTABLE_SCHO2_3[2].s2Value_X := st_SCHO2_KM_GR3;
masTABLE_SCHO2_3[3].s2Value_X := st_SCHO2_SA_AVT_GR3;
masTABLE_SCHO2_3[4].s2Value_X := st_SCHO2_SA_RUCH_GR3;
(* Отображение состояния *)
IF K152_1SHA1_SCHO2_QF3 THEN
	st_SCHO2_QF3 := ' Включено ';
	masTABLE_SCHO2_3[1].dwFillColorAlarm := 16#00FF00;
ELSE
	st_SCHO2_QF3 := ' Выключено ';
	masTABLE_SCHO2_3[1].dwFillColorAlarm := 16#FFFFEF;
END_IF

IF K152_1SHA1_SCHO2_KM_GR3 THEN
	st_SCHO2_KM_GR3 := ' Включено ';
	masTABLE_SCHO2_3[2].dwFillColorAlarm := 16#00FF00;
ELSE
	st_SCHO2_KM_GR3 := ' Выключено ';
	masTABLE_SCHO2_3[2].dwFillColorAlarm := 16#FFFFEF;
END_IF

IF K152_1SHA1_SCHO2_SA_AVT_GR3 THEN
	st_SCHO2_SA_AVT_GR3 := ' Включено ';
	masTABLE_SCHO2_3[3].dwFillColorAlarm := 16#00FF00;
ELSE
	st_SCHO2_SA_AVT_GR3 := ' Выключено ';
	masTABLE_SCHO2_3[3].dwFillColorAlarm := 16#FFFFEF;
END_IF

IF K152_1SHA1_SCHO2_SA_RUCH_GR3 THEN
	st_SCHO2_SA_RUCH_GR3 := ' Включено ';
	masTABLE_SCHO2_3[4].dwFillColorAlarm := 16#00FF00;
ELSE
	st_SCHO2_SA_RUCH_GR3 := ' Выключено ';
	masTABLE_SCHO2_3[4].dwFillColorAlarm := 16#FFFFEF;
END_IF

(* Управление освещением гр.3 *)
rt_bK152_1SHA1_SCHO2_LIGHT_GR3_ON		( CLK := bK152_1SHA1_SCHO2_LIGHT_GR3_ON );
rt_bK152_1SHA1_SCHO2_LIGHT_GR3_OFF		( CLK := bK152_1SHA1_SCHO2_LIGHT_GR3_OFF );

IF rt_bK152_1SHA1_SCHO2_LIGHT_GR3_ON.Q THEN
	bK152_1SHA1_SCHO2_LIGHT_GR3_OFF := FALSE;
	K152_1SHA1_SCHO2_LIGHT_GR3 := TRUE;
ELSIF rt_bK152_1SHA1_SCHO2_LIGHT_GR3_OFF.Q THEN
	bK152_1SHA1_SCHO2_LIGHT_GR3_ON := FALSE;
	K152_1SHA1_SCHO2_LIGHT_GR3 := FALSE;
END_IF


(* ОСВЕЩЕНИЕ ГРУППА 4 *)
(* Столбец 1 *)
masTABLE_SCHO2_4[1].s1Positioin := ' Автоматический выключатель QF4 ';
masTABLE_SCHO2_4[2].s1Positioin := ' Положение магнитного пускателя ';
masTABLE_SCHO2_4[3].s1Positioin := ' Положение переключателя в режиме АВТ. ';
masTABLE_SCHO2_4[4].s1Positioin := ' Положение переключателя в режиме РУЧ. ';
(* Столбец 2 *)
masTABLE_SCHO2_4[1].s2Value_X := st_SCHO2_QF4;
masTABLE_SCHO2_4[2].s2Value_X := st_SCHO2_KM_GR4;
masTABLE_SCHO2_4[3].s2Value_X := st_SCHO2_SA_AVT_GR4;
masTABLE_SCHO2_4[4].s2Value_X := st_SCHO2_SA_RUCH_GR4;
(* Отображение состояния *)
IF K152_1SHA1_SCHO2_QF4 THEN
	st_SCHO2_QF4 := ' Включено ';
	masTABLE_SCHO2_4[1].dwFillColorAlarm := 16#00FF00;
ELSE
	st_SCHO2_QF4 := ' Выключено ';
	masTABLE_SCHO2_4[1].dwFillColorAlarm := 16#FFFFEF;
END_IF

IF K152_1SHA1_SCHO2_KM_GR4 THEN
	st_SCHO2_KM_GR4 := ' Включено ';
	masTABLE_SCHO2_4[2].dwFillColorAlarm := 16#00FF00;
ELSE
	st_SCHO2_KM_GR4 := ' Выключено ';
	masTABLE_SCHO2_4[2].dwFillColorAlarm := 16#FFFFEF;
END_IF

IF K152_1SHA1_SCHO2_SA_AVT_GR4 THEN
	st_SCHO2_SA_AVT_GR4 := ' Включено ';
	masTABLE_SCHO2_4[3].dwFillColorAlarm := 16#00FF00;
ELSE
	st_SCHO2_SA_AVT_GR4 := ' Выключено ';
	masTABLE_SCHO2_4[3].dwFillColorAlarm := 16#FFFFEF;
END_IF

IF K152_1SHA1_SCHO2_SA_RUCH_GR4 THEN
	st_SCHO2_SA_RUCH_GR4 := ' Включено ';
	masTABLE_SCHO2_4[4].dwFillColorAlarm := 16#00FF00;
ELSE
	st_SCHO2_SA_RUCH_GR4 := ' Выключено ';
	masTABLE_SCHO2_4[4].dwFillColorAlarm := 16#FFFFEF;
END_IF

(* Управление освещением гр.4 *)
rt_bK152_1SHA1_SCHO2_LIGHT_GR4_ON		( CLK := bK152_1SHA1_SCHO2_LIGHT_GR4_ON );
rt_bK152_1SHA1_SCHO2_LIGHT_GR4_OFF		( CLK := bK152_1SHA1_SCHO2_LIGHT_GR4_OFF );

IF rt_bK152_1SHA1_SCHO2_LIGHT_GR4_ON.Q THEN
	bK152_1SHA1_SCHO2_LIGHT_GR4_OFF := FALSE;
	K152_1SHA1_SCHO2_LIGHT_GR4 := TRUE;
ELSIF rt_bK152_1SHA1_SCHO2_LIGHT_GR4_OFF.Q THEN
	bK152_1SHA1_SCHO2_LIGHT_GR4_ON := FALSE;
	K152_1SHA1_SCHO2_LIGHT_GR4 := FALSE;
END_IF


(* ОСВЕЩЕНИЕ ГРУППА 5 *)
(* Столбец 1 *)
masTABLE_SCHO2_5[1].s1Positioin := ' Автоматический выключатель QF5 ';
masTABLE_SCHO2_5[2].s1Positioin := ' Положение магнитного пускателя ';
masTABLE_SCHO2_5[3].s1Positioin := ' Положение переключателя в режиме АВТ. ';
masTABLE_SCHO2_5[4].s1Positioin := ' Положение переключателя в режиме РУЧ. ';
(* Столбец 2 *)
masTABLE_SCHO2_5[1].s2Value_X := st_SCHO2_QF5;
masTABLE_SCHO2_5[2].s2Value_X := st_SCHO2_KM_GR5;
masTABLE_SCHO2_5[3].s2Value_X := st_SCHO2_SA_AVT_GR5;
masTABLE_SCHO2_5[4].s2Value_X := st_SCHO2_SA_RUCH_GR5;
(* Отображение состояния *)
IF K152_1SHA1_SCHO2_QF5 THEN
	st_SCHO2_QF5 := ' Включено ';
	masTABLE_SCHO2_5[1].dwFillColorAlarm := 16#00FF00;
ELSE
	st_SCHO2_QF5 := ' Выключено ';
	masTABLE_SCHO2_5[1].dwFillColorAlarm := 16#FFFFEF;
END_IF

IF K152_1SHA1_SCHO2_KM_GR5 THEN
	st_SCHO2_KM_GR5 := ' Включено ';
	masTABLE_SCHO2_5[2].dwFillColorAlarm := 16#00FF00;
ELSE
	st_SCHO2_KM_GR5 := ' Выключено ';
	masTABLE_SCHO2_5[2].dwFillColorAlarm := 16#FFFFEF;
END_IF

IF K152_1SHA1_SCHO2_SA_AVT_GR5 THEN
	st_SCHO2_SA_AVT_GR5 := ' Включено ';
	masTABLE_SCHO2_5[3].dwFillColorAlarm := 16#00FF00;
ELSE
	st_SCHO2_SA_AVT_GR5 := ' Выключено ';
	masTABLE_SCHO2_5[3].dwFillColorAlarm := 16#FFFFEF;
END_IF

IF K152_1SHA1_SCHO2_SA_RUCH_GR5 THEN
	st_SCHO2_SA_RUCH_GR5 := ' Включено ';
	masTABLE_SCHO2_5[4].dwFillColorAlarm := 16#00FF00;
ELSE
	st_SCHO2_SA_RUCH_GR5 := ' Выключено ';
	masTABLE_SCHO2_5[4].dwFillColorAlarm := 16#FFFFEF;
END_IF

(* Управление освещением гр.5 *)
rt_bK152_1SHA1_SCHO2_LIGHT_GR5_ON		( CLK := bK152_1SHA1_SCHO2_LIGHT_GR5_ON );
rt_bK152_1SHA1_SCHO2_LIGHT_GR5_OFF		( CLK := bK152_1SHA1_SCHO2_LIGHT_GR5_OFF );

IF rt_bK152_1SHA1_SCHO2_LIGHT_GR5_ON.Q THEN
	bK152_1SHA1_SCHO2_LIGHT_GR5_OFF := FALSE;
	K152_1SHA1_SCHO2_LIGHT_GR5 := TRUE;
ELSIF rt_bK152_1SHA1_SCHO2_LIGHT_GR5_OFF.Q THEN
	bK152_1SHA1_SCHO2_LIGHT_GR5_ON := FALSE;
	K152_1SHA1_SCHO2_LIGHT_GR5 := FALSE;
END_IF


(* ОСВЕЩЕНИЕ ГРУППА 9 *)
(* Столбец 1 *)
masTABLE_SCHO2_9[1].s1Positioin := ' Автоматический выключатель QF9 ';
masTABLE_SCHO2_9[2].s1Positioin := ' Положение магнитного пускателя ';
masTABLE_SCHO2_9[3].s1Positioin := ' Положение переключателя в режиме АВТ. ';
masTABLE_SCHO2_9[4].s1Positioin := ' Положение переключателя в режиме РУЧ. ';
(* Столбец 2 *)
masTABLE_SCHO2_9[1].s2Value_X := st_SCHO2_QF9;
masTABLE_SCHO2_9[2].s2Value_X := st_SCHO2_KM_GR9;
masTABLE_SCHO2_9[3].s2Value_X := st_SCHO2_SA_AVT_GR9;
masTABLE_SCHO2_9[4].s2Value_X := st_SCHO2_SA_RUCH_GR9;
(* Отображение состояния *)
IF K152_1SHA1_SCHO2_QF9 THEN
	st_SCHO2_QF9 := ' Включено ';
	masTABLE_SCHO2_9[1].dwFillColorAlarm := 16#00FF00;
ELSE
	st_SCHO2_QF9 := ' Выключено ';
	masTABLE_SCHO2_9[1].dwFillColorAlarm := 16#FFFFEF;
END_IF

IF K152_1SHA1_SCHO2_KM_GR9 THEN
	st_SCHO2_KM_GR9 := ' Включено ';
	masTABLE_SCHO2_9[2].dwFillColorAlarm := 16#00FF00;
ELSE
	st_SCHO2_KM_GR9 := ' Выключено ';
	masTABLE_SCHO2_9[2].dwFillColorAlarm := 16#FFFFEF;
END_IF

IF K152_1SHA1_SCHO2_SA_AVT_GR9 THEN
	st_SCHO2_SA_AVT_GR9 := ' Включено ';
	masTABLE_SCHO2_9[3].dwFillColorAlarm := 16#00FF00;
ELSE
	st_SCHO2_SA_AVT_GR9 := ' Выключено ';
	masTABLE_SCHO2_9[3].dwFillColorAlarm := 16#FFFFEF;
END_IF

IF K152_1SHA1_SCHO2_SA_RUCH_GR9 THEN
	st_SCHO2_SA_RUCH_GR9 := ' Включено ';
	masTABLE_SCHO2_9[4].dwFillColorAlarm := 16#00FF00;
ELSE
	st_SCHO2_SA_RUCH_GR9 := ' Выключено ';
	masTABLE_SCHO2_9[4].dwFillColorAlarm := 16#FFFFEF;
END_IF

(* Управление освещением гр.9 *)
rt_bK152_1SHA1_SCHO2_LIGHT_GR9_ON		( CLK := bK152_1SHA1_SCHO2_LIGHT_GR9_ON );
rt_bK152_1SHA1_SCHO2_LIGHT_GR9_OFF		( CLK := bK152_1SHA1_SCHO2_LIGHT_GR9_OFF );

IF rt_bK152_1SHA1_SCHO2_LIGHT_GR9_ON.Q THEN
	bK152_1SHA1_SCHO2_LIGHT_GR9_OFF := FALSE;
	K152_1SHA1_SCHO2_LIGHT_GR9 := TRUE;
ELSIF rt_bK152_1SHA1_SCHO2_LIGHT_GR9_OFF.Q THEN
	bK152_1SHA1_SCHO2_LIGHT_GR9_ON := FALSE;
	K152_1SHA1_SCHO2_LIGHT_GR9 := FALSE;
END_IF
END_PROGRAM

(* POU SCHO2_TABLE_OF_WEEKLY_SCHEDULE, ST *)
PROGRAM SCHO2_TABLE_OF_WEEKLY_SCHEDULE
VAR
	rt_K152_1SHA1_SCHO2_GR1_bMode_AVT 				: R_TRIG;		(* Режим автоматического управления Группой 1 *)
	rt_K152_1SHA1_SCHO2_GR2_bMode_AVT 				: R_TRIG;		(* Режим автоматического управления Группой 2 *)
	rt_K152_1SHA1_SCHO2_GR3_bMode_AVT 				: R_TRIG;		(* Режим автоматического управления Группой 3 *)
	rt_K152_1SHA1_SCHO2_GR4_bMode_AVT 				: R_TRIG;		(* Режим автоматического управления Группой 4 *)
	rt_K152_1SHA1_SCHO2_GR5_bMode_AVT 				: R_TRIG;		(* Режим автоматического управления Группой 5 *)
	rt_K152_1SHA1_SCHO2_GR9_bMode_AVT 				: R_TRIG;		(* Режим автоматического управления Группой 9 *)

	rt_K152_1SHA1_SCHO2_GR1_bMode_MU	 			: R_TRIG;		(* Режим ручного управления Группой 1 *)
	rt_K152_1SHA1_SCHO2_GR2_bMode_MU	 			: R_TRIG;		(* Режим ручного управления Группой 2 *)
	rt_K152_1SHA1_SCHO2_GR3_bMode_MU	 			: R_TRIG;		(* Режим ручного управления Группой 3 *)
	rt_K152_1SHA1_SCHO2_GR4_bMode_MU	 			: R_TRIG;		(* Режим ручного управления Группой 4 *)
	rt_K152_1SHA1_SCHO2_GR5_bMode_MU	 			: R_TRIG;		(* Режим ручного управления Группой 5 *)
	rt_K152_1SHA1_SCHO2_GR9_bMode_MU	 			: R_TRIG;		(* Режим ручного управления Группой 9 *)

END_VAR
(* ---------- ГРУППА 1 ---------- *)
(* Невидимость кнопок выбора режима работы *)
IF K152_1SHA1_SCHO2_GR1_bMode THEN
	Invisible_GR1_bMode := FALSE;
ELSE
	Invisible_GR1_bMode := TRUE;
END_IF

(* Невидимость кнопок вкл/выкл освещения *)
IF K152_1SHA1_SCHO2_GR1_bMode_MU THEN
	Invisible_GR1_bMode_MU := FALSE;
ELSE
	Invisible_GR1_bMode_MU := TRUE;
END_IF

rt_K152_1SHA1_SCHO2_GR1_bMode_AVT (CLK := K152_1SHA1_SCHO2_GR1_bMode_AVT );
rt_K152_1SHA1_SCHO2_GR1_bMode_MU (CLK := K152_1SHA1_SCHO2_GR1_bMode_MU );

(* Отображение режима работы *)
IF rt_K152_1SHA1_SCHO2_GR1_bMode_AVT.Q THEN
	K152_1SHA1_SCHO2_GR1_bMode_MU := FALSE;
	K152_1SHA1_SCHO2_GR1_Mode := ' Автомат ';
END_IF
IF rt_K152_1SHA1_SCHO2_GR1_bMode_MU.Q THEN
	K152_1SHA1_SCHO2_GR1_bMode_AVT := FALSE;
	K152_1SHA1_SCHO2_GR1_Mode := ' Ручной ';
END_IF

(* Столбец "Параметры" *)
masTABLE_WEEKLY_SCHO2_GR1[1].Parameters 	:= ' Время включения ';
masTABLE_WEEKLY_SCHO2_GR1[2].Parameters 	:= ' Время выключения ';

(*	Управление освещением по недельному графику *)
IF K152_1SHA1_SCHO2_GR1_bMode_AVT THEN
	IF Day_of_Today = ' Пн ' THEN
		IF masTABLE_WEEKLY_SCHO2_GR1[1].s1Mon = stTime_graphic THEN
			bK152_1SHA1_SCHO2_LIGHT_GR1_ON := TRUE;
		END_IF
		IF masTABLE_WEEKLY_SCHO2_GR1[2].s1Mon = stTime_graphic THEN
			bK152_1SHA1_SCHO2_LIGHT_GR1_OFF := TRUE;
		END_IF
	ELSIF Day_of_Today = ' Вт ' THEN
		IF masTABLE_WEEKLY_SCHO2_GR1[1].s2Tues = stTime_graphic THEN
			bK152_1SHA1_SCHO2_LIGHT_GR1_ON := TRUE;
		END_IF
		IF masTABLE_WEEKLY_SCHO2_GR1[2].s2Tues = stTime_graphic THEN
			bK152_1SHA1_SCHO2_LIGHT_GR1_OFF := TRUE;
		END_IF
	ELSIF Day_of_Today = ' Ср ' THEN
		IF masTABLE_WEEKLY_SCHO2_GR1[1].s3Wed = stTime_graphic THEN
			bK152_1SHA1_SCHO2_LIGHT_GR1_ON := TRUE;
		END_IF
		IF masTABLE_WEEKLY_SCHO2_GR1[2].s3Wed = stTime_graphic THEN
			bK152_1SHA1_SCHO2_LIGHT_GR1_OFF := TRUE;
		END_IF
	ELSIF Day_of_Today = ' Чт ' THEN
		IF masTABLE_WEEKLY_SCHO2_GR1[1].s4Thrus = stTime_graphic THEN
			bK152_1SHA1_SCHO2_LIGHT_GR1_ON := TRUE;
		END_IF
		IF masTABLE_WEEKLY_SCHO2_GR1[2].s4Thrus = stTime_graphic THEN
			bK152_1SHA1_SCHO2_LIGHT_GR1_OFF := TRUE;
		END_IF
	ELSIF Day_of_Today = ' Пт ' THEN
		IF masTABLE_WEEKLY_SCHO2_GR1[1].s5Fri = stTime_graphic THEN
			bK152_1SHA1_SCHO2_LIGHT_GR1_ON := TRUE;
		END_IF
		IF masTABLE_WEEKLY_SCHO2_GR1[2].s5Fri = stTime_graphic THEN
			bK152_1SHA1_SCHO2_LIGHT_GR1_OFF := TRUE;
		END_IF
	ELSIF Day_of_Today = ' Сб ' THEN
		IF masTABLE_WEEKLY_SCHO2_GR1[1].s6Sat = stTime_graphic THEN
			bK152_1SHA1_SCHO2_LIGHT_GR1_ON := TRUE;
		END_IF
		IF masTABLE_WEEKLY_SCHO2_GR1[2].s6Sat = stTime_graphic THEN
			bK152_1SHA1_SCHO2_LIGHT_GR1_OFF := TRUE;
		END_IF
	ELSIF Day_of_Today = ' Вс ' THEN
		IF masTABLE_WEEKLY_SCHO2_GR1[1].s7Sun = stTime_graphic THEN
			bK152_1SHA1_SCHO2_LIGHT_GR1_ON := TRUE;
		END_IF
		IF masTABLE_WEEKLY_SCHO2_GR1[2].s7Sun = stTime_graphic THEN
			bK152_1SHA1_SCHO2_LIGHT_GR1_OFF := TRUE;
		END_IF
	END_IF
END_IF
END_PROGRAM

(* POU TABLE_OF_POWER_CIRCUITS, ST *)
PROGRAM TABLE_OF_POWER_CIRCUITS
VAR
END_VAR
(* Столбец 1 *)
masPOWER_CIRCUITS[1].s1Text := 'Наличие напряжения на вводе';
masPOWER_CIRCUITS[2].s1Text := 'Питание клапанов';
masPOWER_CIRCUITS[3].s1Text := 'Контактор КМ1';
masPOWER_CIRCUITS[4].s1Text := 'Контактор КМ2';
masPOWER_CIRCUITS[5].s1Text := 'Работа вентилятора приточной установки П3';
masPOWER_CIRCUITS[6].s1Text := 'Работа циркуляционного насоса Н3';
masPOWER_CIRCUITS[7].s1Text := 'Работа БП';
masPOWER_CIRCUITS[8].s1Text := 'Работа ИБП';
masPOWER_CIRCUITS[9].s1Text := 'Работа от батареи';

(* Столбец 2 *)
IF K1 THEN
	masPOWER_CIRCUITS[1].s2Text := 'Включено';
	masPOWER_CIRCUITS[1].dwFillColorAlarm := 16#00FF00;
ELSE
	masPOWER_CIRCUITS[1].s2Text := 'Выключено';
	masPOWER_CIRCUITS[1].dwFillColorAlarm := 16#FFFFEF;
END_IF

IF K152_2P2_QF8 THEN
	masPOWER_CIRCUITS[2].s2Text := 'Включено';
	masPOWER_CIRCUITS[2].dwFillColorAlarm := 16#00FF00;
ELSE
	masPOWER_CIRCUITS[2].s2Text := 'Выключено';
	masPOWER_CIRCUITS[2].dwFillColorAlarm := 16#FFFFEF;
END_IF

IF K152_2P2_KM1 THEN
	masPOWER_CIRCUITS[3].s2Text := 'Включено';
	masPOWER_CIRCUITS[3].dwFillColorAlarm := 16#00FF00;
ELSE
	masPOWER_CIRCUITS[3].s2Text := 'Выключено';
	masPOWER_CIRCUITS[3].dwFillColorAlarm := 16#FFFFEF;
END_IF
IF K152_2P2_KM2 THEN
	masPOWER_CIRCUITS[4].s2Text := 'Включено';
	masPOWER_CIRCUITS[4].dwFillColorAlarm := 16#00FF00;
ELSE
	masPOWER_CIRCUITS[4].s2Text := 'Выключено';
	masPOWER_CIRCUITS[4].dwFillColorAlarm := 16#FFFFEF;
END_IF
IF K152_2P2_HL4 THEN
	masPOWER_CIRCUITS[5].s2Text := 'Включено';
	masPOWER_CIRCUITS[5].dwFillColorAlarm := 16#00FF00;
ELSE
	masPOWER_CIRCUITS[5].s2Text := 'Выключено';
	masPOWER_CIRCUITS[5].dwFillColorAlarm := 16#FFFFEF;
END_IF
IF K152_2P2_HL6 THEN
	masPOWER_CIRCUITS[6].s2Text := 'Включено';
	masPOWER_CIRCUITS[6].dwFillColorAlarm := 16#00FF00;
ELSE
	masPOWER_CIRCUITS[6].s2Text := 'Выключено';
	masPOWER_CIRCUITS[6].dwFillColorAlarm := 16#FFFFEF;
END_IF
IF K152_2P2_WORK_BP THEN
	masPOWER_CIRCUITS[7].s2Text := 'Включено';
	masPOWER_CIRCUITS[7].dwFillColorAlarm := 16#00FF00;
ELSE
	masPOWER_CIRCUITS[7].s2Text := 'Выключено';
	masPOWER_CIRCUITS[7].dwFillColorAlarm := 16#FFFFEF;
END_IF
IF K152_2P2_WORK_IBP THEN
	masPOWER_CIRCUITS[8].s2Text := 'Включено';
	masPOWER_CIRCUITS[8].dwFillColorAlarm := 16#00FF00;
ELSE
	masPOWER_CIRCUITS[8].s2Text := 'Выключено';
	masPOWER_CIRCUITS[8].dwFillColorAlarm := 16#FFFFEF;
END_IF
IF K152_2P2_WORK_OF_BATTERY THEN
	masPOWER_CIRCUITS[9].s2Text := 'Включено';
	masPOWER_CIRCUITS[9].dwFillColorAlarm := 16#00FF00;
ELSE
	masPOWER_CIRCUITS[9].s2Text := 'Выключено';
	masPOWER_CIRCUITS[9].dwFillColorAlarm := 16#FFFFEF;
END_IF
END_PROGRAM

(* Visualisation A0_START_WINDOW
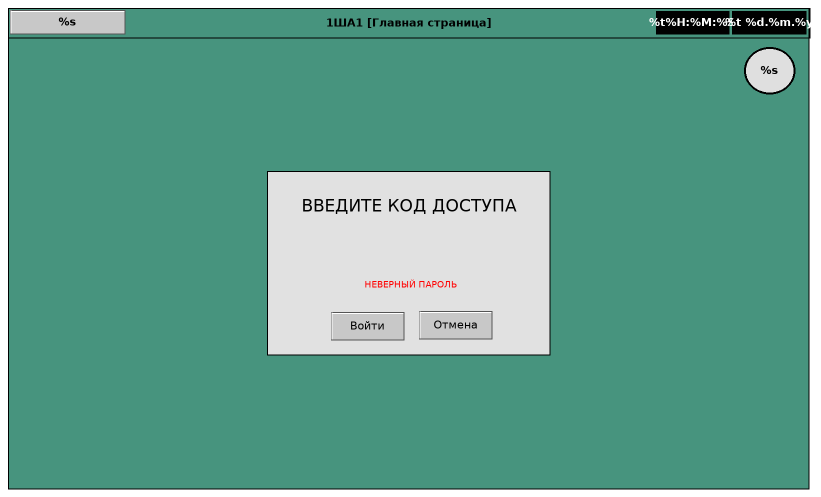
rectangle at (259,163)-(542,347): invisible if VHOD.AUTORIZATION_INVISIBLE
rectangle at (262,176)-(540,219): text "ВВЕДИТЕ КОД ДОСТУПА"; invisible if VHOD.AUTORIZATION_INVISIBLE
button at (323,304)-(396,332): text "Войти"; invisible if VHOD.bOK; opens A1_START_WINDOW
rectangle at (315,267)-(491,286): text "НЕВЕРНЫЙ ПАРОЛЬ"; shows VHOD.FAIL_PASS_TEXT; invisible if VHOD.FAIL_PASS
button at (411,303)-(484,331): text "Отмена"; invisible if VHOD.AUTORIZATION_INVISIBLE; toggles VHOD.bVihod
ellipse at (736,39)-(787,86): text "%s"; shows LAMPS.LAMP_HL1; alarm colour if .K152_1SHA1_HL1
rectangle at (0,0)-(802,30): text "1ША1 [Главная страница]"
rectangle at (648,3)-(721,26): text "%t%H:%M:%S"
rectangle at (724,3)-(798,26): text "%t %d.%m.%y"
button at (2,2)-(117,26): text "%s"; shows VHOD.User; taps VHOD.bAUTORIZATION
1 more shapes without text or variables
1 elements of other kinds (tables, trends, ...) not read
*)

(* Visualisation A1_START_WINDOW
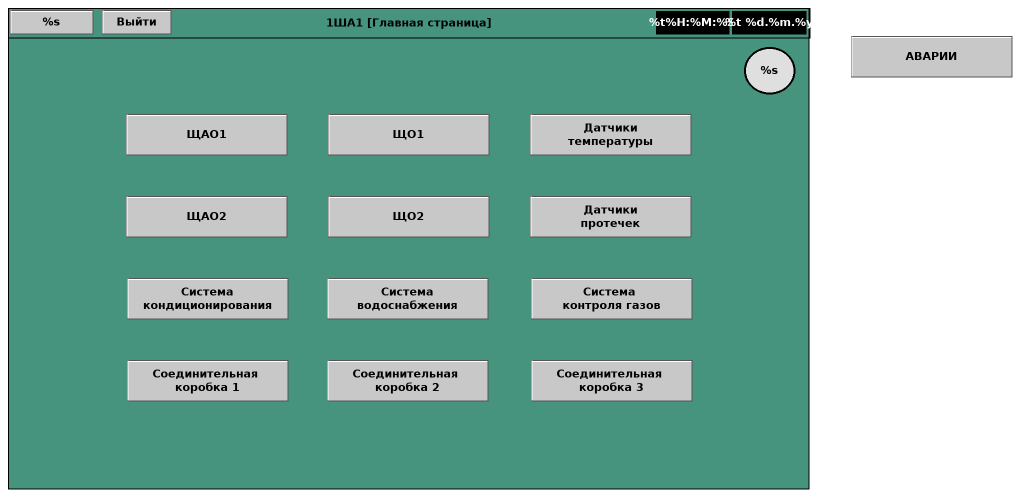
button at (118,106)-(279,147): text "ЩАО1"; opens SCHAO1
button at (320,106)-(481,147): text "ЩО1"; opens SCHO1
ellipse at (736,39)-(787,86): text "%s"; shows LAMPS.LAMP_HL1; alarm colour if .K152_1SHA1_HL1
button at (118,188)-(279,229): text "ЩАО2"; opens SCHAO2
button at (522,188)-(683,229): text "Датчики / протечек"; opens PROTECHKI_CONTROL
button at (320,188)-(481,229): text "ЩО2"; opens SCHO2
button at (319,270)-(480,311): text "Система / водоснабжения"; opens SYSTEM_WATER_SUPPLY
rectangle at (0,0)-(802,30): text "1ША1 [Главная страница]"
button at (2,2)-(85,26): text "%s"; shows VHOD.User; taps VHOD.bAUTORIZATION
button at (522,106)-(683,147): text "Датчики / температуры"; opens TEMP_CONTROL
button at (94,2)-(163,26): text "Выйти"; toggles VHOD.bVihod; opens A0_START_WINDOW
rectangle at (648,3)-(721,26): text "%t%H:%M:%S"
rectangle at (724,3)-(798,26): text "%t %d.%m.%y"
button at (119,270)-(280,311): text "Система / кондиционирования"; opens SYSTEM_CONDITIONING
button at (523,270)-(684,311): text "Система / контроля газов"; opens SYSTEM_GAS_CONTROL
button at (319,352)-(480,393): text "Соединительная / коробка 2"; opens KC2
button at (119,352)-(280,393): text "Соединительная / коробка 1"; opens KC1
button at (523,352)-(684,393): text "Соединительная / коробка 3"; opens KC3
button at (843,28)-(1004,69): text "АВАРИИ"; opens ALARM
1 more shapes without text or variables
1 elements of other kinds (tables, trends, ...) not read
*)

(* Visualisation ALARM
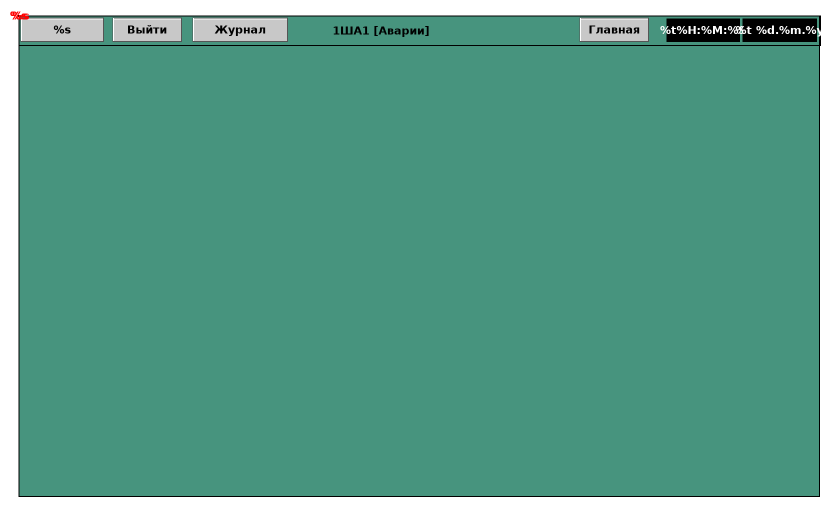
rectangle at (0,0)-(802,30): text "1ША1 [Аварии]"
button at (2,2)-(85,26): text "%s"; shows VHOD.User
button at (94,2)-(163,26): text "Выйти"; toggles VHOD.bVihod; opens A0_START_WINDOW
button at (561,2)-(630,26): text "Главная"; opens A1_START_WINDOW
rectangle at (0,0)-(0,0): text "%s"; shows ALARM_TABLE[INDEX].s1Date
rectangle at (0,0)-(0,0): text "%s"; shows ALARM_TABLE[INDEX].s2Time
rectangle at (0,0)-(0,0): text "%s"; shows ALARM_TABLE[INDEX].s3Text
button at (174,2)-(269,26): text "Журнал"; opens ALARM_JOUNAL
rectangle at (648,3)-(721,26): text "%t%H:%M:%S"
rectangle at (724,3)-(798,26): text "%t %d.%m.%y"
1 more shapes without text or variables
*)

(* Visualisation ALARM_JOUNAL
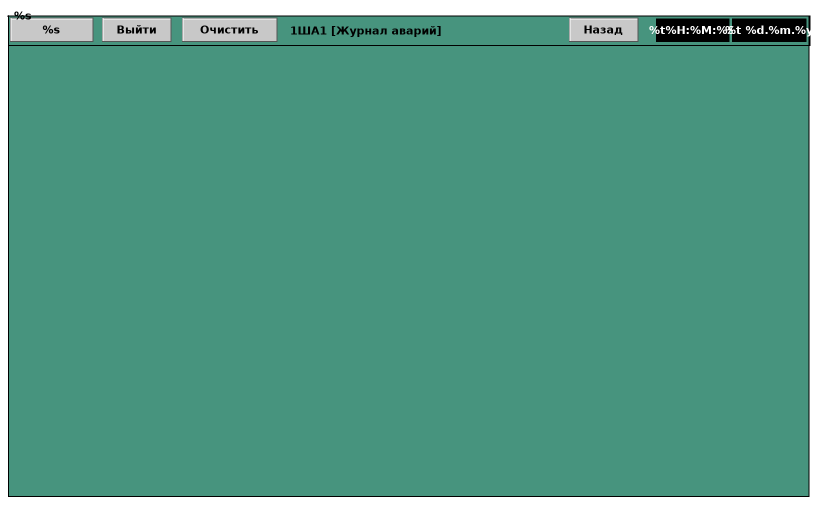
rectangle at (0,0)-(802,30): text "1ША1 [Журнал аварий]"
button at (2,2)-(85,26): text "%s"; shows VHOD.User
button at (94,2)-(163,26): text "Выйти"; toggles VHOD.bVihod; opens A0_START_WINDOW
button at (561,2)-(630,26): text "Назад"; opens ALARM
rectangle at (0,0)-(0,0): text "%s"; shows ALARM_DATA[INDEX]
button at (174,2)-(269,26): text "Очистить"; taps .bClearAlarmData
rectangle at (648,3)-(721,26): text "%t%H:%M:%S"
rectangle at (724,3)-(798,26): text "%t %d.%m.%y"
1 more shapes without text or variables
*)

(* Visualisation KC1
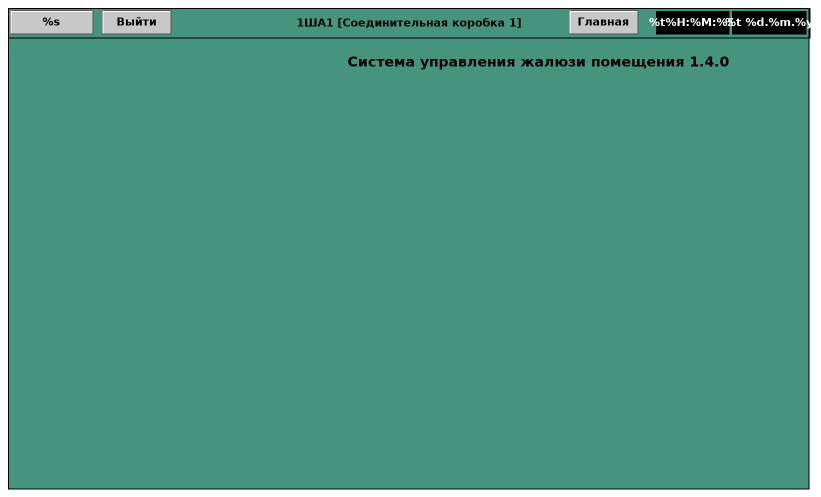
rectangle at (0,0)-(802,30): text "1ША1 [Соединительная коробка 1]"
button at (2,2)-(85,26): text "%s"; shows VHOD.User
button at (94,2)-(163,26): text "Выйти"; toggles VHOD.bVihod; opens A0_START_WINDOW
button at (561,2)-(630,26): text "Главная"; opens A1_START_WINDOW
rectangle at (648,3)-(721,26): text "%t%H:%M:%S"
rectangle at (724,3)-(798,26): text "%t %d.%m.%y"
rectangle at (233,42)-(828,65): text "Система управления жалюзи помещения 1.4.0"
1 more shapes without text or variables
*)

(* Visualisation KC2
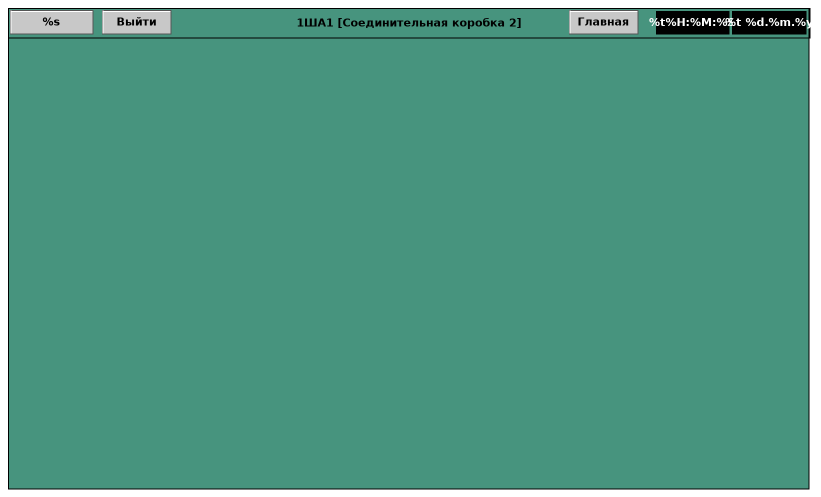
rectangle at (0,0)-(802,30): text "1ША1 [Соединительная коробка 2]"
button at (2,2)-(85,26): text "%s"; shows VHOD.User
button at (94,2)-(163,26): text "Выйти"; toggles VHOD.bVihod; opens A0_START_WINDOW
button at (561,2)-(630,26): text "Главная"; opens A1_START_WINDOW
rectangle at (648,3)-(721,26): text "%t%H:%M:%S"
rectangle at (724,3)-(798,26): text "%t %d.%m.%y"
1 more shapes without text or variables
*)

(* Visualisation KC3
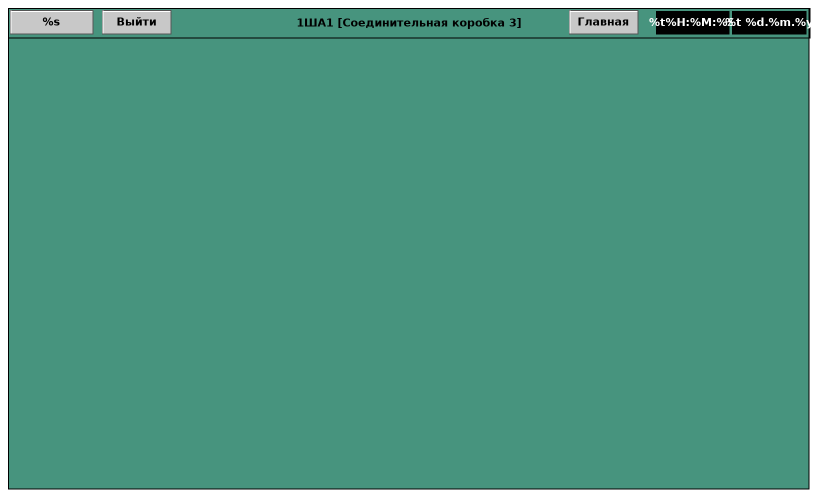
rectangle at (0,0)-(802,30): text "1ША1 [Соединительная коробка 3]"
button at (2,2)-(85,26): text "%s"; shows VHOD.User
button at (94,2)-(163,26): text "Выйти"; toggles VHOD.bVihod; opens A0_START_WINDOW
button at (561,2)-(630,26): text "Главная"; opens A1_START_WINDOW
rectangle at (648,3)-(721,26): text "%t%H:%M:%S"
rectangle at (724,3)-(798,26): text "%t %d.%m.%y"
1 more shapes without text or variables
*)

(* Visualisation POWER_CIRCUITS
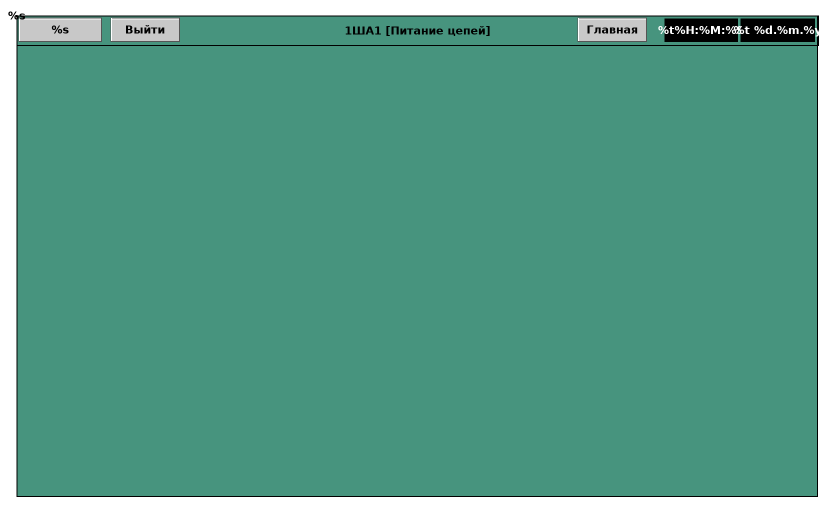
rectangle at (0,0)-(802,30): text "1ША1 [Питание цепей]"
button at (2,2)-(85,26): text "%s"; shows VHOD.User
button at (94,2)-(163,26): text "Выйти"; toggles VHOD.bVihod; opens A0_START_WINDOW
button at (561,2)-(630,26): text "Главная"; opens A1_START_WINDOW
rectangle at (0,0)-(0,0): text "%s"; shows masTABLE_POWER[INDEX].s1Text
rectangle at (648,3)-(721,26): text "%t%H:%M:%S"
rectangle at (724,3)-(798,26): text "%t %d.%m.%y"
1 more shapes without text or variables
*)

(* Visualisation PROTECHKI_CONTROL
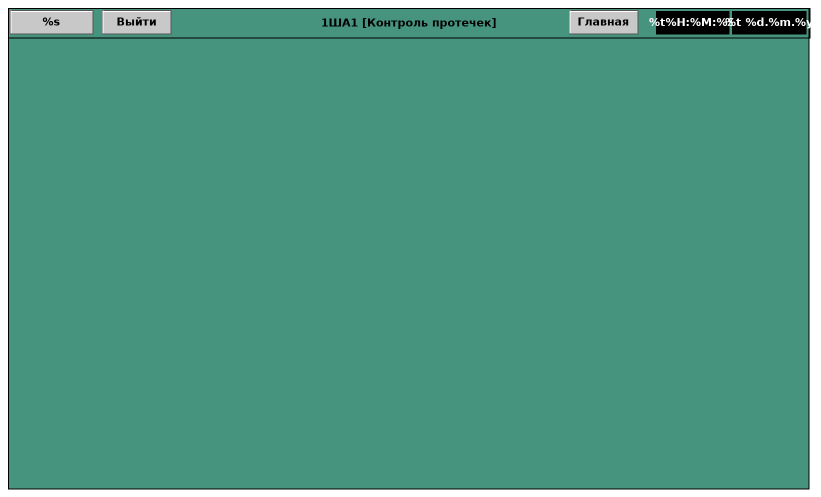
rectangle at (0,0)-(802,30): text "1ША1 [Контроль протечек]"
button at (2,2)-(85,26): text "%s"; shows VHOD.User
button at (94,2)-(163,26): text "Выйти"; toggles VHOD.bVihod; opens A0_START_WINDOW
button at (561,2)-(630,26): text "Главная"; opens A1_START_WINDOW
rectangle at (648,3)-(721,26): text "%t%H:%M:%S"
rectangle at (724,3)-(798,26): text "%t %d.%m.%y"
1 more shapes without text or variables
1 elements of other kinds (tables, trends, ...) not read
*)

(* Visualisation SCHAO1
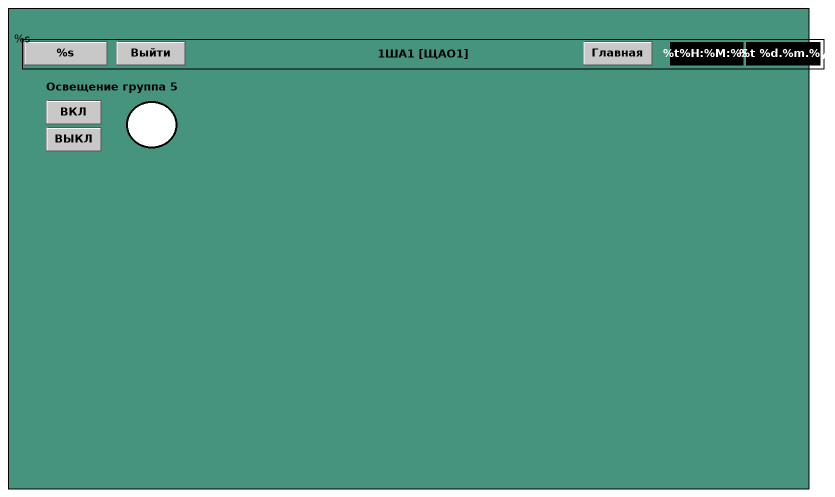
rectangle at (0,0)-(802,30): text "1ША1 [ЩАО1]"
button at (2,2)-(85,26): text "%s"; shows VHOD.User
button at (94,2)-(163,26): text "Выйти"; toggles VHOD.bVihod; opens A0_START_WINDOW
button at (561,2)-(630,26): text "Главная"; opens A1_START_WINDOW
rectangle at (648,3)-(721,26): text "%t%H:%M:%S"
rectangle at (724,3)-(798,26): text "%t %d.%m.%y"
rectangle at (0,0)-(0,0): text "%s"; shows masTABLE_SCHAO1[INDEX].On_Off; alarm colour if masTABLE_SCHAO1[INDEX].ON; editable
rectangle at (4,36)-(176,60): text "Освещение группа 5"
button at (24,61)-(79,85): text "ВКЛ"; toggles .bK152_1SHA1_SCHAO1_LIGHT_GR5_ON
button at (24,88)-(79,112): text "ВЫКЛ"; taps .bK152_1SHA1_SCHAO1_LIGHT_GR5_OFF
ellipse at (104,62)-(155,109): alarm colour if .K152_1SHA1_SCHAO1_LIGHT_GR5
1 more shapes without text or variables
1 elements of other kinds (tables, trends, ...) not read
*)

(* Visualisation SCHAO2
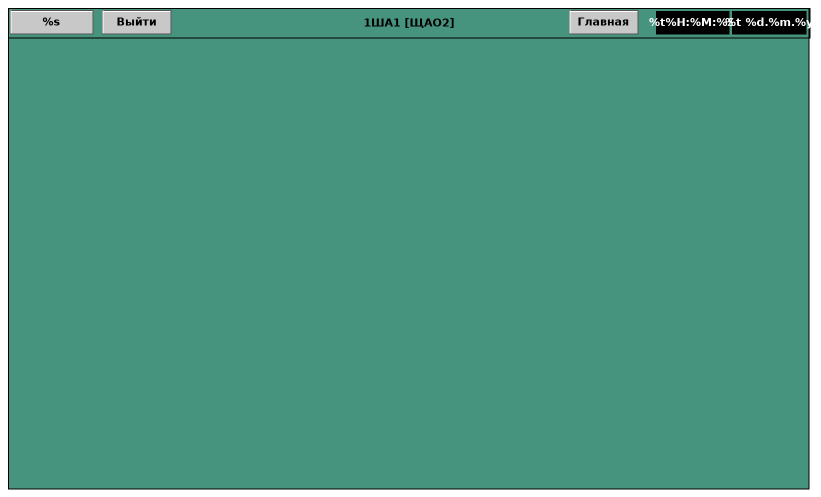
rectangle at (0,0)-(802,30): text "1ША1 [ЩАО2]"
button at (2,2)-(85,26): text "%s"; shows VHOD.User
button at (94,2)-(163,26): text "Выйти"; toggles VHOD.bVihod; opens A0_START_WINDOW
button at (561,2)-(630,26): text "Главная"; opens A1_START_WINDOW
rectangle at (648,3)-(721,26): text "%t%H:%M:%S"
rectangle at (724,3)-(798,26): text "%t %d.%m.%y"
1 more shapes without text or variables
*)

(* Visualisation SCHO1
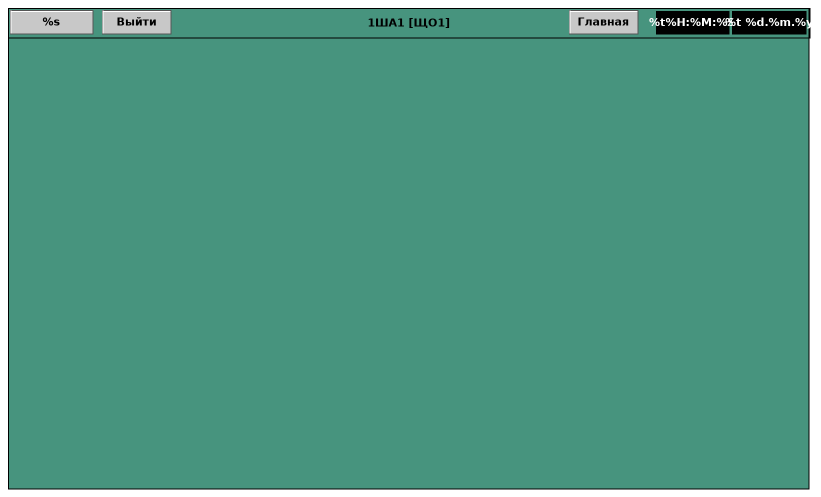
rectangle at (0,0)-(802,30): text "1ША1 [ЩО1]"
button at (2,2)-(85,26): text "%s"; shows VHOD.User
button at (94,2)-(163,26): text "Выйти"; toggles VHOD.bVihod; opens A0_START_WINDOW
button at (561,2)-(630,26): text "Главная"; opens A1_START_WINDOW
rectangle at (648,3)-(721,26): text "%t%H:%M:%S"
rectangle at (724,3)-(798,26): text "%t %d.%m.%y"
1 more shapes without text or variables
*)

(* Visualisation SCHO2
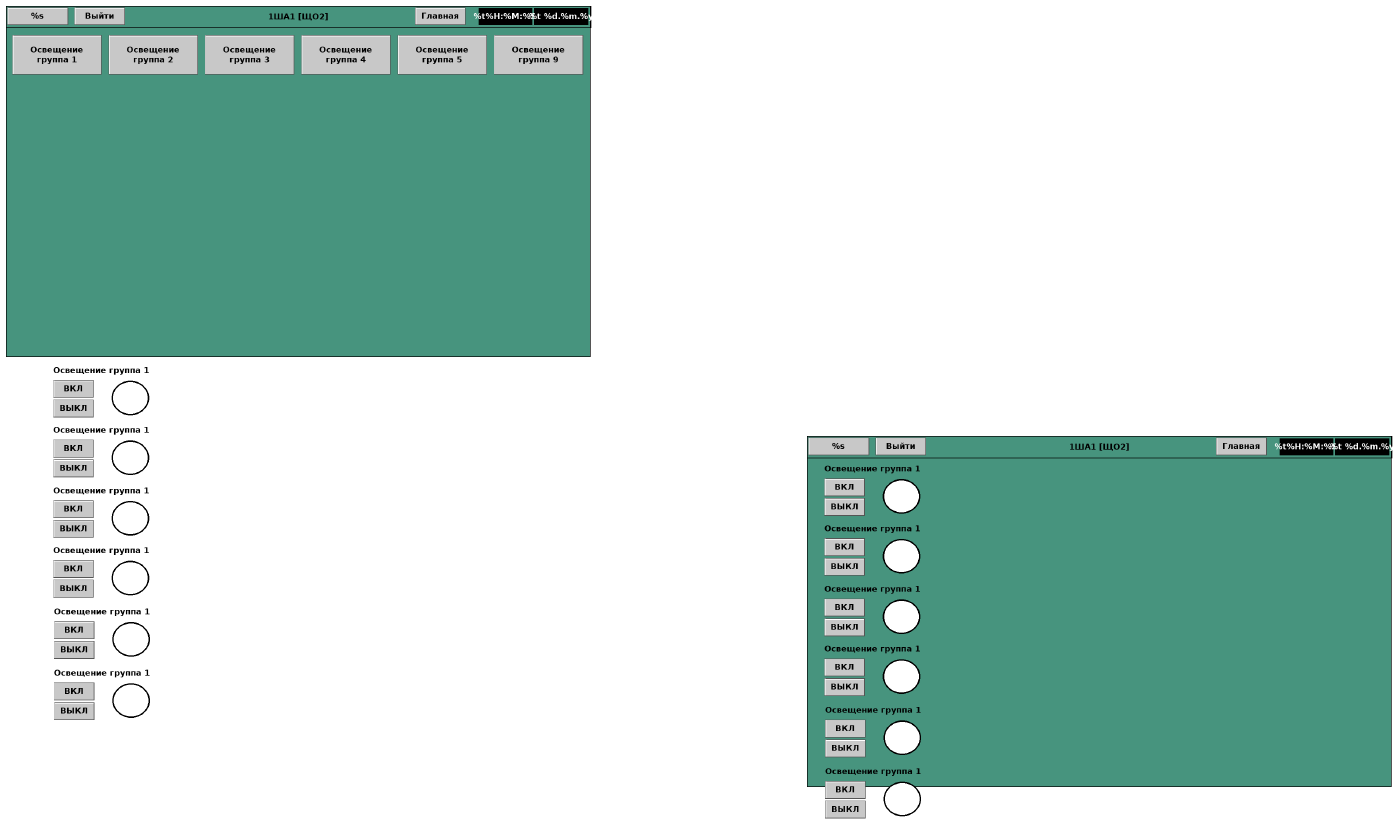
rectangle at (0,0)-(802,30): text "1ША1 [ЩО2]"
button at (2,2)-(85,26): text "%s"; shows VHOD.User
button at (94,2)-(163,26): text "Выйти"; toggles VHOD.bVihod; opens A0_START_WINDOW
button at (561,2)-(630,26): text "Главная"; opens A1_START_WINDOW
rectangle at (648,3)-(721,26): text "%t%H:%M:%S"
rectangle at (724,3)-(798,26): text "%t %d.%m.%y"
rectangle at (45,488)-(217,512): text "Освещение группа 1"
button at (65,513)-(120,537): text "ВКЛ"; toggles .bK152_1SHA1_SCHAO1_LIGHT_GR5_ON
button at (65,540)-(120,564): text "ВЫКЛ"; taps .bK152_1SHA1_SCHAO1_LIGHT_GR5_OFF
ellipse at (145,514)-(196,561): alarm colour if .K152_1SHA1_SCHAO1_LIGHT_GR5
rectangle at (45,570)-(217,594): text "Освещение группа 1"
button at (65,595)-(120,619): text "ВКЛ"; toggles .bK152_1SHA1_SCHAO1_LIGHT_GR5_ON
button at (65,622)-(120,646): text "ВЫКЛ"; taps .bK152_1SHA1_SCHAO1_LIGHT_GR5_OFF
ellipse at (145,596)-(196,643): alarm colour if .K152_1SHA1_SCHAO1_LIGHT_GR5
rectangle at (45,653)-(217,677): text "Освещение группа 1"
button at (65,678)-(120,702): text "ВКЛ"; toggles .bK152_1SHA1_SCHAO1_LIGHT_GR5_ON
button at (65,705)-(120,729): text "ВЫКЛ"; taps .bK152_1SHA1_SCHAO1_LIGHT_GR5_OFF
ellipse at (145,679)-(196,726): alarm colour if .K152_1SHA1_SCHAO1_LIGHT_GR5
rectangle at (45,735)-(217,759): text "Освещение группа 1"
button at (65,760)-(120,784): text "ВКЛ"; toggles .bK152_1SHA1_SCHAO1_LIGHT_GR5_ON
button at (65,787)-(120,811): text "ВЫКЛ"; taps .bK152_1SHA1_SCHAO1_LIGHT_GR5_OFF
ellipse at (145,761)-(196,808): alarm colour if .K152_1SHA1_SCHAO1_LIGHT_GR5
rectangle at (46,819)-(218,843): text "Освещение группа 1"
button at (66,844)-(121,868): text "ВКЛ"; toggles .bK152_1SHA1_SCHAO1_LIGHT_GR5_ON
button at (66,871)-(121,895): text "ВЫКЛ"; taps .bK152_1SHA1_SCHAO1_LIGHT_GR5_OFF
ellipse at (146,845)-(197,892): alarm colour if .K152_1SHA1_SCHAO1_LIGHT_GR5
rectangle at (46,903)-(218,927): text "Освещение группа 1"
button at (66,928)-(121,952): text "ВКЛ"; toggles .bK152_1SHA1_SCHAO1_LIGHT_GR5_ON
button at (66,955)-(121,979): text "ВЫКЛ"; taps .bK152_1SHA1_SCHAO1_LIGHT_GR5_OFF
ellipse at (146,929)-(197,976): alarm colour if .K152_1SHA1_SCHAO1_LIGHT_GR5
rectangle at (1098,590)-(1900,620): text "1ША1 [ЩО2]"
button at (1100,592)-(1183,616): text "%s"; shows VHOD.User
button at (1192,592)-(1261,616): text "Выйти"; toggles VHOD.bVihod; opens A0_START_WINDOW
button at (1659,592)-(1728,616): text "Главная"; opens A1_START_WINDOW
rectangle at (1746,593)-(1819,616): text "%t%H:%M:%S"
rectangle at (1822,593)-(1896,616): text "%t %d.%m.%y"
rectangle at (1102,623)-(1274,647): text "Освещение группа 1"
button at (1122,648)-(1177,672): text "ВКЛ"; toggles .bK152_1SHA1_SCHAO1_LIGHT_GR5_ON
button at (1122,675)-(1177,699): text "ВЫКЛ"; taps .bK152_1SHA1_SCHAO1_LIGHT_GR5_OFF
ellipse at (1202,649)-(1253,696): alarm colour if .K152_1SHA1_SCHAO1_LIGHT_GR5
rectangle at (1102,705)-(1274,729): text "Освещение группа 1"
button at (1122,730)-(1177,754): text "ВКЛ"; toggles .bK152_1SHA1_SCHAO1_LIGHT_GR5_ON
button at (1122,757)-(1177,781): text "ВЫКЛ"; taps .bK152_1SHA1_SCHAO1_LIGHT_GR5_OFF
ellipse at (1202,731)-(1253,778): alarm colour if .K152_1SHA1_SCHAO1_LIGHT_GR5
rectangle at (1102,788)-(1274,812): text "Освещение группа 1"
button at (1122,813)-(1177,837): text "ВКЛ"; toggles .bK152_1SHA1_SCHAO1_LIGHT_GR5_ON
button at (1122,840)-(1177,864): text "ВЫКЛ"; taps .bK152_1SHA1_SCHAO1_LIGHT_GR5_OFF
ellipse at (1202,814)-(1253,861): alarm colour if .K152_1SHA1_SCHAO1_LIGHT_GR5
rectangle at (1102,870)-(1274,894): text "Освещение группа 1"
button at (1122,895)-(1177,919): text "ВКЛ"; toggles .bK152_1SHA1_SCHAO1_LIGHT_GR5_ON
button at (1122,922)-(1177,946): text "ВЫКЛ"; taps .bK152_1SHA1_SCHAO1_LIGHT_GR5_OFF
ellipse at (1202,896)-(1253,943): alarm colour if .K152_1SHA1_SCHAO1_LIGHT_GR5
rectangle at (1103,954)-(1275,978): text "Освещение группа 1"
button at (1123,979)-(1178,1003): text "ВКЛ"; toggles .bK152_1SHA1_SCHAO1_LIGHT_GR5_ON
button at (1123,1006)-(1178,1030): text "ВЫКЛ"; taps .bK152_1SHA1_SCHAO1_LIGHT_GR5_OFF
ellipse at (1203,980)-(1254,1027): alarm colour if .K152_1SHA1_SCHAO1_LIGHT_GR5
rectangle at (1103,1038)-(1275,1062): text "Освещение группа 1"
button at (1123,1063)-(1178,1087): text "ВКЛ"; toggles .bK152_1SHA1_SCHAO1_LIGHT_GR5_ON
button at (1123,1090)-(1178,1114): text "ВЫКЛ"; taps .bK152_1SHA1_SCHAO1_LIGHT_GR5_OFF
ellipse at (1203,1064)-(1254,1111): alarm colour if .K152_1SHA1_SCHAO1_LIGHT_GR5
button at (9,40)-(131,94): text "Освещение / группа 1"; opens SCHO2_GR1
button at (141,40)-(263,94): text "Освещение / группа 2"; opens SCHO2_GR2
button at (273,40)-(395,94): text "Освещение / группа 3"; opens SCHO2_GR3
button at (405,40)-(527,94): text "Освещение / группа 4"; opens SCHO2_GR4
button at (537,40)-(659,94): text "Освещение / группа 5"; opens SCHO2_GR5
button at (669,40)-(791,94): text "Освещение / группа 9"; opens SCHO2_GR9
2 more shapes without text or variables
16 elements of other kinds (tables, trends, ...) not read
*)

(* Visualisation SCHO2_GR1
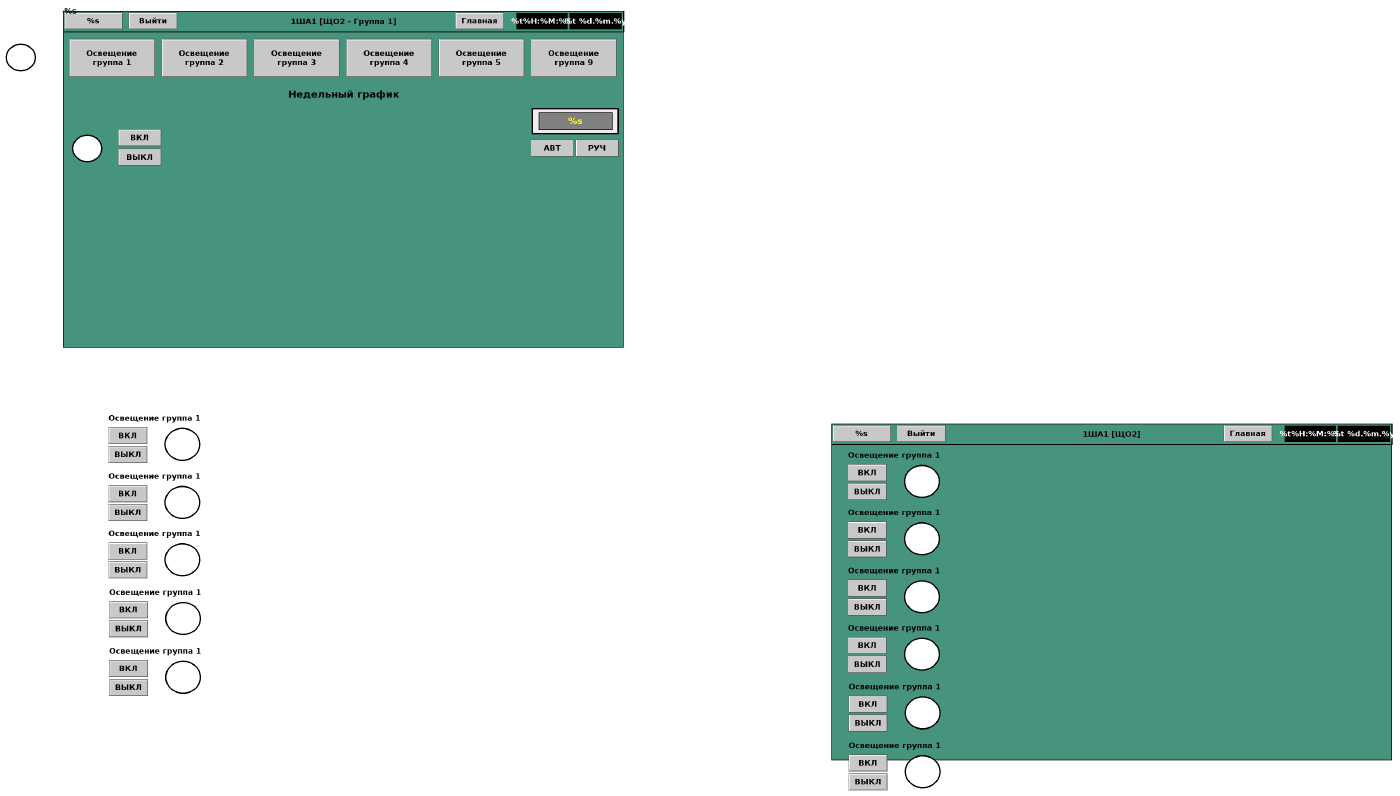
button at (669,184)-(730,208): text "АВТ"; invisible if .Invisible_GR1_bMode; toggles .K152_1SHA1_SCHO2_GR1_bMode_AVT
rectangle at (0,0)-(802,30): text "1ША1 [ЩО2 - Группа 1]"
button at (2,2)-(85,26): text "%s"; shows VHOD.User
button at (94,2)-(163,26): text "Выйти"; toggles VHOD.bVihod; opens A0_START_WINDOW
button at (561,2)-(630,26): text "Главная"; opens A1_START_WINDOW
rectangle at (648,3)-(721,26): text "%t%H:%M:%S"
rectangle at (724,3)-(798,26): text "%t %d.%m.%y"
rectangle at (148,107)-(655,131): text "Недельный график"
button at (79,169)-(140,193): text "ВКЛ"; invisible if .Invisible_GR1_bMode_MU; toggles .bK152_1SHA1_SCHO2_LIGHT_GR1_ON
button at (79,197)-(140,221): text "ВЫКЛ"; invisible if .Invisible_GR1_bMode_MU; toggles .bK152_1SHA1_SCHO2_LIGHT_GR1_OFF
ellipse at (13,177)-(56,216): alarm colour if .K152_1SHA1_SCHO2_KM_GR1
rectangle at (45,570)-(217,594): text "Освещение группа 1"
button at (65,595)-(120,619): text "ВКЛ"; toggles .bK152_1SHA1_SCHAO1_LIGHT_GR5_ON
button at (65,622)-(120,646): text "ВЫКЛ"; taps .bK152_1SHA1_SCHAO1_LIGHT_GR5_OFF
ellipse at (145,596)-(196,643): alarm colour if .K152_1SHA1_SCHAO1_LIGHT_GR5
rectangle at (45,653)-(217,677): text "Освещение группа 1"
button at (65,678)-(120,702): text "ВКЛ"; toggles .bK152_1SHA1_SCHAO1_LIGHT_GR5_ON
button at (65,705)-(120,729): text "ВЫКЛ"; taps .bK152_1SHA1_SCHAO1_LIGHT_GR5_OFF
ellipse at (145,679)-(196,726): alarm colour if .K152_1SHA1_SCHAO1_LIGHT_GR5
rectangle at (45,735)-(217,759): text "Освещение группа 1"
button at (65,760)-(120,784): text "ВКЛ"; toggles .bK152_1SHA1_SCHAO1_LIGHT_GR5_ON
button at (65,787)-(120,811): text "ВЫКЛ"; taps .bK152_1SHA1_SCHAO1_LIGHT_GR5_OFF
ellipse at (145,761)-(196,808): alarm colour if .K152_1SHA1_SCHAO1_LIGHT_GR5
rectangle at (46,819)-(218,843): text "Освещение группа 1"
button at (66,844)-(121,868): text "ВКЛ"; toggles .bK152_1SHA1_SCHAO1_LIGHT_GR5_ON
button at (66,871)-(121,895): text "ВЫКЛ"; taps .bK152_1SHA1_SCHAO1_LIGHT_GR5_OFF
ellipse at (146,845)-(197,892): alarm colour if .K152_1SHA1_SCHAO1_LIGHT_GR5
rectangle at (46,903)-(218,927): text "Освещение группа 1"
button at (66,928)-(121,952): text "ВКЛ"; toggles .bK152_1SHA1_SCHAO1_LIGHT_GR5_ON
button at (66,955)-(121,979): text "ВЫКЛ"; taps .bK152_1SHA1_SCHAO1_LIGHT_GR5_OFF
ellipse at (146,929)-(197,976): alarm colour if .K152_1SHA1_SCHAO1_LIGHT_GR5
rectangle at (1098,590)-(1900,620): text "1ША1 [ЩО2]"
button at (1100,592)-(1183,616): text "%s"; shows VHOD.User
button at (1192,592)-(1261,616): text "Выйти"; toggles VHOD.bVihod; opens A0_START_WINDOW
button at (1659,592)-(1728,616): text "Главная"; opens A1_START_WINDOW
rectangle at (1746,593)-(1819,616): text "%t%H:%M:%S"
rectangle at (1822,593)-(1896,616): text "%t %d.%m.%y"
rectangle at (1102,623)-(1274,647): text "Освещение группа 1"
button at (1122,648)-(1177,672): text "ВКЛ"; toggles .bK152_1SHA1_SCHAO1_LIGHT_GR5_ON
button at (1122,675)-(1177,699): text "ВЫКЛ"; taps .bK152_1SHA1_SCHAO1_LIGHT_GR5_OFF
ellipse at (1202,649)-(1253,696): alarm colour if .K152_1SHA1_SCHAO1_LIGHT_GR5
rectangle at (1102,705)-(1274,729): text "Освещение группа 1"
button at (1122,730)-(1177,754): text "ВКЛ"; toggles .bK152_1SHA1_SCHAO1_LIGHT_GR5_ON
button at (1122,757)-(1177,781): text "ВЫКЛ"; taps .bK152_1SHA1_SCHAO1_LIGHT_GR5_OFF
ellipse at (1202,731)-(1253,778): alarm colour if .K152_1SHA1_SCHAO1_LIGHT_GR5
rectangle at (1102,788)-(1274,812): text "Освещение группа 1"
button at (1122,813)-(1177,837): text "ВКЛ"; toggles .bK152_1SHA1_SCHAO1_LIGHT_GR5_ON
button at (1122,840)-(1177,864): text "ВЫКЛ"; taps .bK152_1SHA1_SCHAO1_LIGHT_GR5_OFF
ellipse at (1202,814)-(1253,861): alarm colour if .K152_1SHA1_SCHAO1_LIGHT_GR5
rectangle at (1102,870)-(1274,894): text "Освещение группа 1"
button at (1122,895)-(1177,919): text "ВКЛ"; toggles .bK152_1SHA1_SCHAO1_LIGHT_GR5_ON
button at (1122,922)-(1177,946): text "ВЫКЛ"; taps .bK152_1SHA1_SCHAO1_LIGHT_GR5_OFF
ellipse at (1202,896)-(1253,943): alarm colour if .K152_1SHA1_SCHAO1_LIGHT_GR5
rectangle at (1103,954)-(1275,978): text "Освещение группа 1"
button at (1123,979)-(1178,1003): text "ВКЛ"; toggles .bK152_1SHA1_SCHAO1_LIGHT_GR5_ON
button at (1123,1006)-(1178,1030): text "ВЫКЛ"; taps .bK152_1SHA1_SCHAO1_LIGHT_GR5_OFF
ellipse at (1203,980)-(1254,1027): alarm colour if .K152_1SHA1_SCHAO1_LIGHT_GR5
rectangle at (1103,1038)-(1275,1062): text "Освещение группа 1"
button at (1123,1063)-(1178,1087): text "ВКЛ"; toggles .bK152_1SHA1_SCHAO1_LIGHT_GR5_ON
button at (1123,1090)-(1178,1114): text "ВЫКЛ"; taps .bK152_1SHA1_SCHAO1_LIGHT_GR5_OFF
ellipse at (1203,1064)-(1254,1111): alarm colour if .K152_1SHA1_SCHAO1_LIGHT_GR5
button at (9,40)-(131,94): text "Освещение / группа 1"; opens SCHO2_GR1
button at (141,40)-(263,94): text "Освещение / группа 2"; opens SCHO2_GR2
button at (273,40)-(395,94): text "Освещение / группа 3"; opens SCHO2_GR3
button at (405,40)-(527,94): text "Освещение / группа 4"; opens SCHO2_GR4
button at (537,40)-(659,94): text "Освещение / группа 5"; opens SCHO2_GR5
button at (669,40)-(791,94): text "Освещение / группа 9"; opens SCHO2_GR9
button at (733,184)-(794,208): text "РУЧ"; invisible if .Invisible_GR1_bMode; toggles .K152_1SHA1_SCHO2_GR1_bMode_MU
rounded rectangle at (680,145)-(785,170): text "%s"; shows .K152_1SHA1_SCHO2_GR1_Mode; toggles .K152_1SHA1_SCHO2_GR1_bMode
rectangle at (0,0)-(0,0): text "%s"; shows masTABLE_WEEKLY_SCHO2_GR1[INDEX].Parameters
ellipse at (-82,47)-(-39,86): alarm colour if .K152_1SHA1_SCHO2_LIGHT_GR1
3 more shapes without text or variables
15 elements of other kinds (tables, trends, ...) not read
*)

(* Visualisation SCHO2_GR2
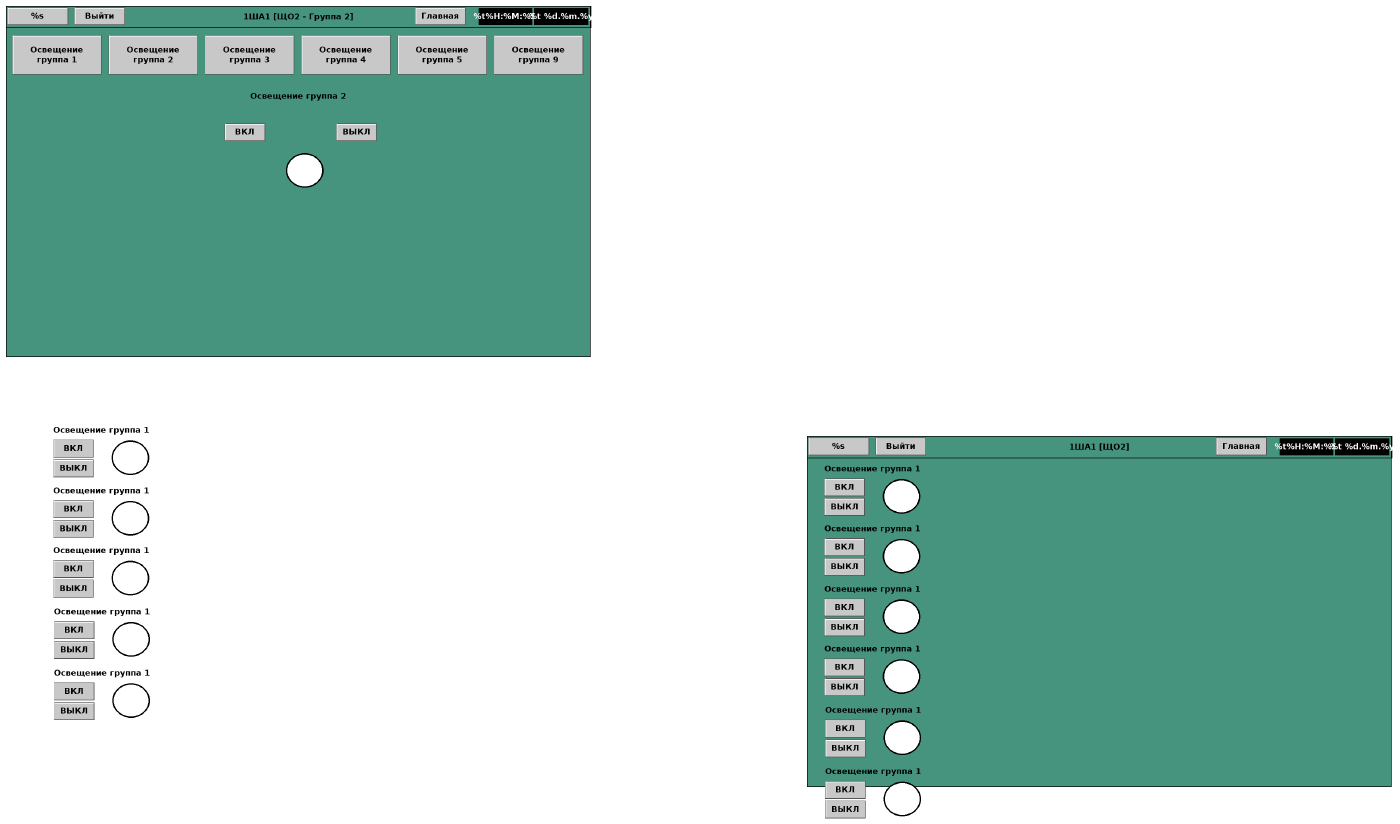
rectangle at (0,0)-(802,30): text "1ША1 [ЩО2 - Группа 2]"
button at (2,2)-(85,26): text "%s"; shows VHOD.User
button at (94,2)-(163,26): text "Выйти"; toggles VHOD.bVihod; opens A0_START_WINDOW
button at (561,2)-(630,26): text "Главная"; opens A1_START_WINDOW
rectangle at (648,3)-(721,26): text "%t%H:%M:%S"
rectangle at (724,3)-(798,26): text "%t %d.%m.%y"
rectangle at (6,107)-(796,141): text "Освещение группа 2"
button at (300,161)-(355,185): text "ВКЛ"; toggles .bK152_1SHA1_SCHO2_LIGHT_GR2_ON
button at (453,161)-(508,185): text "ВЫКЛ"; taps .bK152_1SHA1_SCHO2_LIGHT_GR2_OFF
ellipse at (384,202)-(435,249): alarm colour if .K152_1SHA1_SCHO2_KM_GR2
rectangle at (45,570)-(217,594): text "Освещение группа 1"
button at (65,595)-(120,619): text "ВКЛ"; toggles .bK152_1SHA1_SCHAO1_LIGHT_GR5_ON
button at (65,622)-(120,646): text "ВЫКЛ"; taps .bK152_1SHA1_SCHAO1_LIGHT_GR5_OFF
ellipse at (145,596)-(196,643): alarm colour if .K152_1SHA1_SCHAO1_LIGHT_GR5
rectangle at (45,653)-(217,677): text "Освещение группа 1"
button at (65,678)-(120,702): text "ВКЛ"; toggles .bK152_1SHA1_SCHAO1_LIGHT_GR5_ON
button at (65,705)-(120,729): text "ВЫКЛ"; taps .bK152_1SHA1_SCHAO1_LIGHT_GR5_OFF
ellipse at (145,679)-(196,726): alarm colour if .K152_1SHA1_SCHAO1_LIGHT_GR5
rectangle at (45,735)-(217,759): text "Освещение группа 1"
button at (65,760)-(120,784): text "ВКЛ"; toggles .bK152_1SHA1_SCHAO1_LIGHT_GR5_ON
button at (65,787)-(120,811): text "ВЫКЛ"; taps .bK152_1SHA1_SCHAO1_LIGHT_GR5_OFF
ellipse at (145,761)-(196,808): alarm colour if .K152_1SHA1_SCHAO1_LIGHT_GR5
rectangle at (46,819)-(218,843): text "Освещение группа 1"
button at (66,844)-(121,868): text "ВКЛ"; toggles .bK152_1SHA1_SCHAO1_LIGHT_GR5_ON
button at (66,871)-(121,895): text "ВЫКЛ"; taps .bK152_1SHA1_SCHAO1_LIGHT_GR5_OFF
ellipse at (146,845)-(197,892): alarm colour if .K152_1SHA1_SCHAO1_LIGHT_GR5
rectangle at (46,903)-(218,927): text "Освещение группа 1"
button at (66,928)-(121,952): text "ВКЛ"; toggles .bK152_1SHA1_SCHAO1_LIGHT_GR5_ON
button at (66,955)-(121,979): text "ВЫКЛ"; taps .bK152_1SHA1_SCHAO1_LIGHT_GR5_OFF
ellipse at (146,929)-(197,976): alarm colour if .K152_1SHA1_SCHAO1_LIGHT_GR5
rectangle at (1098,590)-(1900,620): text "1ША1 [ЩО2]"
button at (1100,592)-(1183,616): text "%s"; shows VHOD.User
button at (1192,592)-(1261,616): text "Выйти"; toggles VHOD.bVihod; opens A0_START_WINDOW
button at (1659,592)-(1728,616): text "Главная"; opens A1_START_WINDOW
rectangle at (1746,593)-(1819,616): text "%t%H:%M:%S"
rectangle at (1822,593)-(1896,616): text "%t %d.%m.%y"
rectangle at (1102,623)-(1274,647): text "Освещение группа 1"
button at (1122,648)-(1177,672): text "ВКЛ"; toggles .bK152_1SHA1_SCHAO1_LIGHT_GR5_ON
button at (1122,675)-(1177,699): text "ВЫКЛ"; taps .bK152_1SHA1_SCHAO1_LIGHT_GR5_OFF
ellipse at (1202,649)-(1253,696): alarm colour if .K152_1SHA1_SCHAO1_LIGHT_GR5
rectangle at (1102,705)-(1274,729): text "Освещение группа 1"
button at (1122,730)-(1177,754): text "ВКЛ"; toggles .bK152_1SHA1_SCHAO1_LIGHT_GR5_ON
button at (1122,757)-(1177,781): text "ВЫКЛ"; taps .bK152_1SHA1_SCHAO1_LIGHT_GR5_OFF
ellipse at (1202,731)-(1253,778): alarm colour if .K152_1SHA1_SCHAO1_LIGHT_GR5
rectangle at (1102,788)-(1274,812): text "Освещение группа 1"
button at (1122,813)-(1177,837): text "ВКЛ"; toggles .bK152_1SHA1_SCHAO1_LIGHT_GR5_ON
button at (1122,840)-(1177,864): text "ВЫКЛ"; taps .bK152_1SHA1_SCHAO1_LIGHT_GR5_OFF
ellipse at (1202,814)-(1253,861): alarm colour if .K152_1SHA1_SCHAO1_LIGHT_GR5
rectangle at (1102,870)-(1274,894): text "Освещение группа 1"
button at (1122,895)-(1177,919): text "ВКЛ"; toggles .bK152_1SHA1_SCHAO1_LIGHT_GR5_ON
button at (1122,922)-(1177,946): text "ВЫКЛ"; taps .bK152_1SHA1_SCHAO1_LIGHT_GR5_OFF
ellipse at (1202,896)-(1253,943): alarm colour if .K152_1SHA1_SCHAO1_LIGHT_GR5
rectangle at (1103,954)-(1275,978): text "Освещение группа 1"
button at (1123,979)-(1178,1003): text "ВКЛ"; toggles .bK152_1SHA1_SCHAO1_LIGHT_GR5_ON
button at (1123,1006)-(1178,1030): text "ВЫКЛ"; taps .bK152_1SHA1_SCHAO1_LIGHT_GR5_OFF
ellipse at (1203,980)-(1254,1027): alarm colour if .K152_1SHA1_SCHAO1_LIGHT_GR5
rectangle at (1103,1038)-(1275,1062): text "Освещение группа 1"
button at (1123,1063)-(1178,1087): text "ВКЛ"; toggles .bK152_1SHA1_SCHAO1_LIGHT_GR5_ON
button at (1123,1090)-(1178,1114): text "ВЫКЛ"; taps .bK152_1SHA1_SCHAO1_LIGHT_GR5_OFF
ellipse at (1203,1064)-(1254,1111): alarm colour if .K152_1SHA1_SCHAO1_LIGHT_GR5
button at (9,40)-(131,94): text "Освещение / группа 1"; opens SCHO2_GR1
button at (141,40)-(263,94): text "Освещение / группа 2"; opens SCHO2_GR2
button at (273,40)-(395,94): text "Освещение / группа 3"; opens SCHO2_GR3
button at (405,40)-(527,94): text "Освещение / группа 4"; opens SCHO2_GR4
button at (537,40)-(659,94): text "Освещение / группа 5"; opens SCHO2_GR5
button at (669,40)-(791,94): text "Освещение / группа 9"; opens SCHO2_GR9
2 more shapes without text or variables
14 elements of other kinds (tables, trends, ...) not read
*)

(* Visualisation SCHO2_GR3
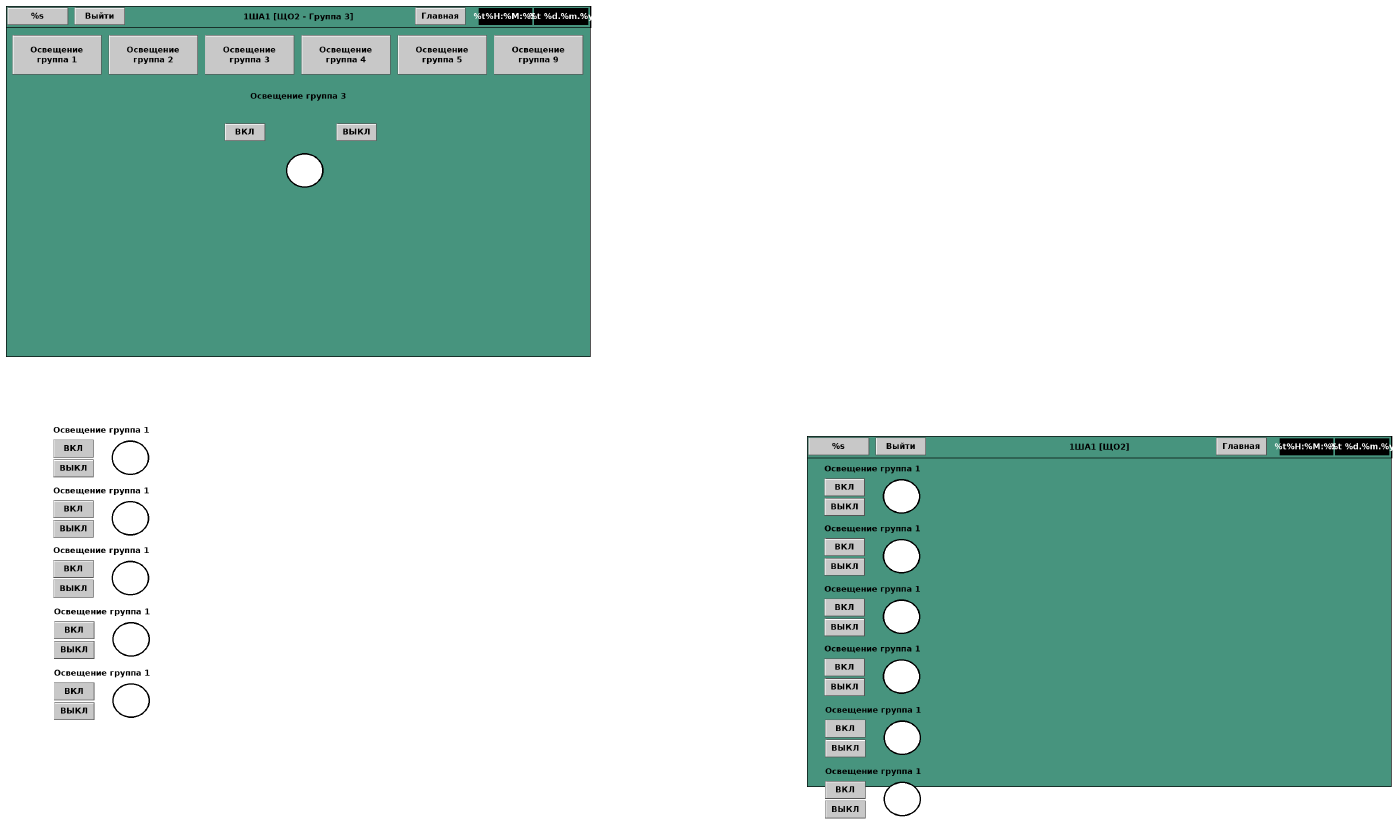
rectangle at (0,0)-(802,30): text "1ША1 [ЩО2 - Группа 3]"
button at (2,2)-(85,26): text "%s"; shows VHOD.User
button at (94,2)-(163,26): text "Выйти"; toggles VHOD.bVihod; opens A0_START_WINDOW
button at (561,2)-(630,26): text "Главная"; opens A1_START_WINDOW
rectangle at (648,3)-(721,26): text "%t%H:%M:%S"
rectangle at (724,3)-(798,26): text "%t %d.%m.%y"
rectangle at (6,107)-(796,141): text "Освещение группа 3"
button at (300,161)-(355,185): text "ВКЛ"; toggles .bK152_1SHA1_SCHO2_LIGHT_GR3_ON
button at (453,161)-(508,185): text "ВЫКЛ"; taps .bK152_1SHA1_SCHO2_LIGHT_GR3_OFF
ellipse at (384,202)-(435,249): alarm colour if .K152_1SHA1_SCHO2_KM_GR3
rectangle at (45,570)-(217,594): text "Освещение группа 1"
button at (65,595)-(120,619): text "ВКЛ"; toggles .bK152_1SHA1_SCHAO1_LIGHT_GR5_ON
button at (65,622)-(120,646): text "ВЫКЛ"; taps .bK152_1SHA1_SCHAO1_LIGHT_GR5_OFF
ellipse at (145,596)-(196,643): alarm colour if .K152_1SHA1_SCHAO1_LIGHT_GR5
rectangle at (45,653)-(217,677): text "Освещение группа 1"
button at (65,678)-(120,702): text "ВКЛ"; toggles .bK152_1SHA1_SCHAO1_LIGHT_GR5_ON
button at (65,705)-(120,729): text "ВЫКЛ"; taps .bK152_1SHA1_SCHAO1_LIGHT_GR5_OFF
ellipse at (145,679)-(196,726): alarm colour if .K152_1SHA1_SCHAO1_LIGHT_GR5
rectangle at (45,735)-(217,759): text "Освещение группа 1"
button at (65,760)-(120,784): text "ВКЛ"; toggles .bK152_1SHA1_SCHAO1_LIGHT_GR5_ON
button at (65,787)-(120,811): text "ВЫКЛ"; taps .bK152_1SHA1_SCHAO1_LIGHT_GR5_OFF
ellipse at (145,761)-(196,808): alarm colour if .K152_1SHA1_SCHAO1_LIGHT_GR5
rectangle at (46,819)-(218,843): text "Освещение группа 1"
button at (66,844)-(121,868): text "ВКЛ"; toggles .bK152_1SHA1_SCHAO1_LIGHT_GR5_ON
button at (66,871)-(121,895): text "ВЫКЛ"; taps .bK152_1SHA1_SCHAO1_LIGHT_GR5_OFF
ellipse at (146,845)-(197,892): alarm colour if .K152_1SHA1_SCHAO1_LIGHT_GR5
rectangle at (46,903)-(218,927): text "Освещение группа 1"
button at (66,928)-(121,952): text "ВКЛ"; toggles .bK152_1SHA1_SCHAO1_LIGHT_GR5_ON
button at (66,955)-(121,979): text "ВЫКЛ"; taps .bK152_1SHA1_SCHAO1_LIGHT_GR5_OFF
ellipse at (146,929)-(197,976): alarm colour if .K152_1SHA1_SCHAO1_LIGHT_GR5
rectangle at (1098,590)-(1900,620): text "1ША1 [ЩО2]"
button at (1100,592)-(1183,616): text "%s"; shows VHOD.User
button at (1192,592)-(1261,616): text "Выйти"; toggles VHOD.bVihod; opens A0_START_WINDOW
button at (1659,592)-(1728,616): text "Главная"; opens A1_START_WINDOW
rectangle at (1746,593)-(1819,616): text "%t%H:%M:%S"
rectangle at (1822,593)-(1896,616): text "%t %d.%m.%y"
rectangle at (1102,623)-(1274,647): text "Освещение группа 1"
button at (1122,648)-(1177,672): text "ВКЛ"; toggles .bK152_1SHA1_SCHAO1_LIGHT_GR5_ON
button at (1122,675)-(1177,699): text "ВЫКЛ"; taps .bK152_1SHA1_SCHAO1_LIGHT_GR5_OFF
ellipse at (1202,649)-(1253,696): alarm colour if .K152_1SHA1_SCHAO1_LIGHT_GR5
rectangle at (1102,705)-(1274,729): text "Освещение группа 1"
button at (1122,730)-(1177,754): text "ВКЛ"; toggles .bK152_1SHA1_SCHAO1_LIGHT_GR5_ON
button at (1122,757)-(1177,781): text "ВЫКЛ"; taps .bK152_1SHA1_SCHAO1_LIGHT_GR5_OFF
ellipse at (1202,731)-(1253,778): alarm colour if .K152_1SHA1_SCHAO1_LIGHT_GR5
rectangle at (1102,788)-(1274,812): text "Освещение группа 1"
button at (1122,813)-(1177,837): text "ВКЛ"; toggles .bK152_1SHA1_SCHAO1_LIGHT_GR5_ON
button at (1122,840)-(1177,864): text "ВЫКЛ"; taps .bK152_1SHA1_SCHAO1_LIGHT_GR5_OFF
ellipse at (1202,814)-(1253,861): alarm colour if .K152_1SHA1_SCHAO1_LIGHT_GR5
rectangle at (1102,870)-(1274,894): text "Освещение группа 1"
button at (1122,895)-(1177,919): text "ВКЛ"; toggles .bK152_1SHA1_SCHAO1_LIGHT_GR5_ON
button at (1122,922)-(1177,946): text "ВЫКЛ"; taps .bK152_1SHA1_SCHAO1_LIGHT_GR5_OFF
ellipse at (1202,896)-(1253,943): alarm colour if .K152_1SHA1_SCHAO1_LIGHT_GR5
rectangle at (1103,954)-(1275,978): text "Освещение группа 1"
button at (1123,979)-(1178,1003): text "ВКЛ"; toggles .bK152_1SHA1_SCHAO1_LIGHT_GR5_ON
button at (1123,1006)-(1178,1030): text "ВЫКЛ"; taps .bK152_1SHA1_SCHAO1_LIGHT_GR5_OFF
ellipse at (1203,980)-(1254,1027): alarm colour if .K152_1SHA1_SCHAO1_LIGHT_GR5
rectangle at (1103,1038)-(1275,1062): text "Освещение группа 1"
button at (1123,1063)-(1178,1087): text "ВКЛ"; toggles .bK152_1SHA1_SCHAO1_LIGHT_GR5_ON
button at (1123,1090)-(1178,1114): text "ВЫКЛ"; taps .bK152_1SHA1_SCHAO1_LIGHT_GR5_OFF
ellipse at (1203,1064)-(1254,1111): alarm colour if .K152_1SHA1_SCHAO1_LIGHT_GR5
button at (9,40)-(131,94): text "Освещение / группа 1"; opens SCHO2_GR1
button at (141,40)-(263,94): text "Освещение / группа 2"; opens SCHO2_GR2
button at (273,40)-(395,94): text "Освещение / группа 3"; opens SCHO2_GR3
button at (405,40)-(527,94): text "Освещение / группа 4"; opens SCHO2_GR4
button at (537,40)-(659,94): text "Освещение / группа 5"; opens SCHO2_GR5
button at (669,40)-(791,94): text "Освещение / группа 9"; opens SCHO2_GR9
2 more shapes without text or variables
14 elements of other kinds (tables, trends, ...) not read
*)

